// TIA Portal V17 export
// export: Created 2025-03-07T09:16:40.4760323Z, ExportSetting WithDefaults, DisplayName Totally Integrated Automation Portal, DisplayVersion V17 Update 8, DisplayName TIA Portal Openness, DisplayVersion V17 Update 8, DisplayName TIA Portal Version Control Interface, DisplayVersion V17, DisplayName SINAMICS Startdrive Advanced, DisplayVersion V17 SP2, DisplayName SINAMICS Startdrive G110M, G120, G120C, G120D, G120P, G115D, DisplayVersion V17 SP2, DisplayName SINAMICS Startdrive G130, G150, S120, S150, SINAMICS MV, S210, DisplayVersion V17 SP2, DisplayName STEP 7 Professional, DisplayVersion V17 Update 8, DisplayName SINUMERIK ONE STEP 7 Toolbox, DisplayVersion V17 Update 12, DisplayName SINUMERIK 840D sl STEP 7 Toolbox, DisplayVersion V17 Update 12, DisplayName STEP 7 Safety, DisplayVersion V17 Update 6, DisplayName WinCC Advanced, DisplayVersion V17 Update 8
FUNCTION "FC2431_FULL_DEPTHS_UNIT_02" : Void   // FC2431, LAD
{ S7_Optimized_Access := 'FALSE' }
AUTHOR : ETXETAR
VERSION : 1.0
// Fixture 1 and Fixture 3 will do Face A
// Fixture 2 and Fixture 4 will do Face B
// stored: AutoNumber false, IsIECCheckEnabled false, SetENOAutomatically false, UDAEnableTagReadback false
   VAR_TEMP   // added for the SCL form of the ladder/FBD networks
      _w1 : Bool;
   END_VAR
BEGIN

REGION Network 1: <<<<<<<<<<<<<<<<<<<<< UNIT 02 >>>>>>>>>>>>>>>>>>>>>
END_REGION

REGION Network 2: <<<<<<<<<<<<<<<<<<<< FIXTURE 1 >>>>>>>>>>>>>>>>>>>>
END_REGION

REGION Network 3: UNIT 02 FIXTURE 1 STATION 1 FULL DEPTH / FULL DEPTH 1 PULSE
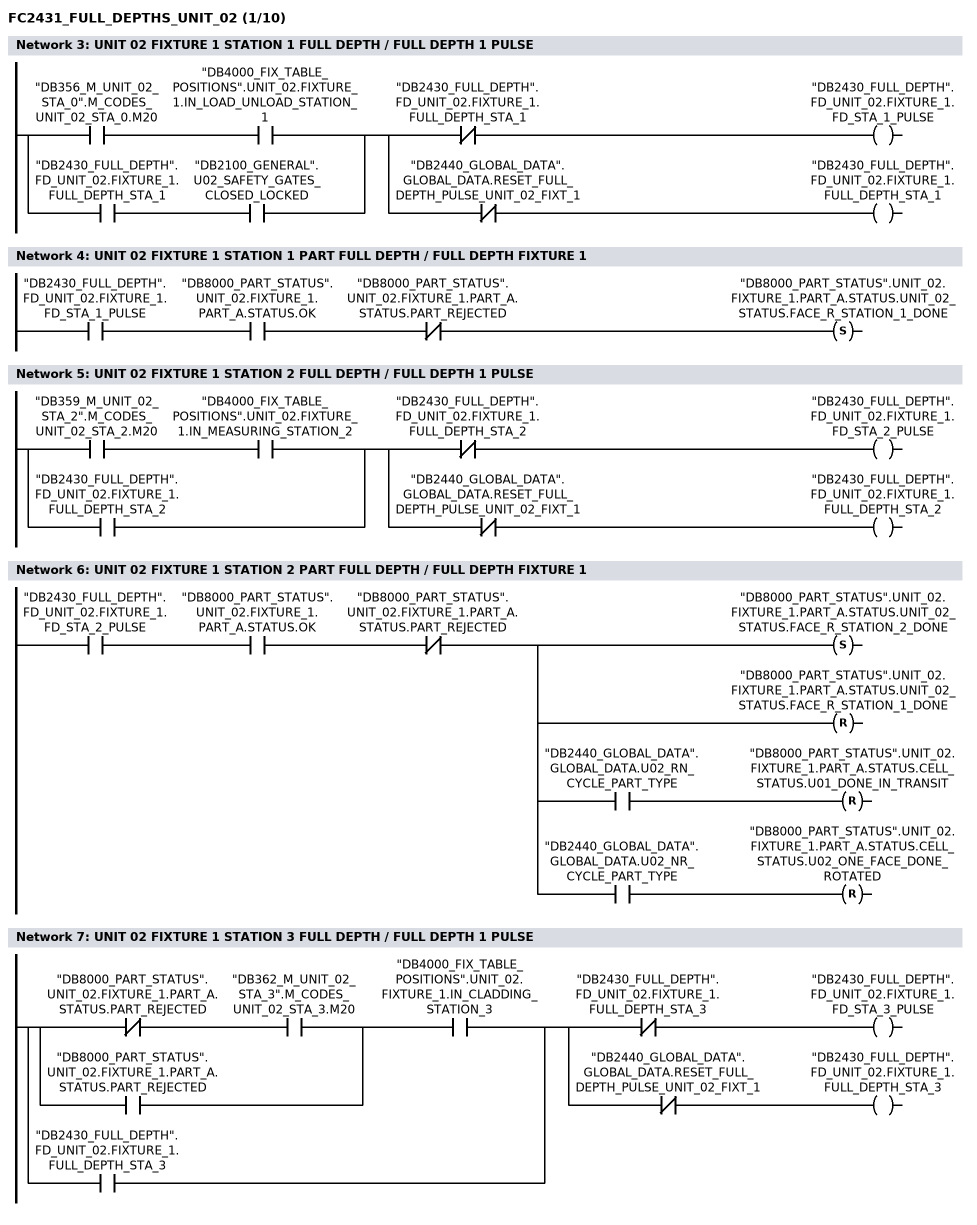
   RUNG wire#powerrail
      Contact( "DB356_M_UNIT_02_STA_0".M_CODES_UNIT_02_STA_0.M20 )
      Contact( "DB4000_FIX_TABLE_POSITIONS".UNIT_02.FIXTURE_1.IN_LOAD_UNLOAD_STATION_1 )
      wire#w1
      I_Contact( "DB2430_FULL_DEPTH".FD_UNIT_02.FIXTURE_1.FULL_DEPTH_STA_1 )
      Coil( "DB2430_FULL_DEPTH".FD_UNIT_02.FIXTURE_1.FD_STA_1_PULSE )
   END_RUNG
   RUNG wire#powerrail
      Contact( "DB2430_FULL_DEPTH".FD_UNIT_02.FIXTURE_1.FULL_DEPTH_STA_1 )
      Contact( "DB2100_GENERAL".U02_SAFETY_GATES_CLOSED_LOCKED )
   END_RUNG wire#w1
   RUNG wire#w1
      I_Contact( "DB2440_GLOBAL_DATA".GLOBAL_DATA.RESET_FULL_DEPTH_PULSE_UNIT_02_FIXT_1 )
      Coil( "DB2430_FULL_DEPTH".FD_UNIT_02.FIXTURE_1.FULL_DEPTH_STA_1 )
   END_RUNG
   // the same network as SCL:
   #_w1 := ("DB356_M_UNIT_02_STA_0".M_CODES_UNIT_02_STA_0.M20 AND "DB4000_FIX_TABLE_POSITIONS".UNIT_02.FIXTURE_1.IN_LOAD_UNLOAD_STATION_1) OR ("DB2430_FULL_DEPTH".FD_UNIT_02.FIXTURE_1.FULL_DEPTH_STA_1 AND "DB2100_GENERAL".U02_SAFETY_GATES_CLOSED_LOCKED);
   "DB2430_FULL_DEPTH".FD_UNIT_02.FIXTURE_1.FD_STA_1_PULSE := #_w1 AND NOT "DB2430_FULL_DEPTH".FD_UNIT_02.FIXTURE_1.FULL_DEPTH_STA_1;
   "DB2430_FULL_DEPTH".FD_UNIT_02.FIXTURE_1.FULL_DEPTH_STA_1 := #_w1 AND NOT "DB2440_GLOBAL_DATA".GLOBAL_DATA.RESET_FULL_DEPTH_PULSE_UNIT_02_FIXT_1;
END_REGION

REGION Network 4: UNIT 02 FIXTURE 1 STATION 1 PART FULL DEPTH / FULL DEPTH FIXTURE 1
   RUNG wire#powerrail
      Contact( "DB2430_FULL_DEPTH".FD_UNIT_02.FIXTURE_1.FD_STA_1_PULSE )
      Contact( "DB8000_PART_STATUS".UNIT_02.FIXTURE_1.PART_A.STATUS.OK )
      I_Contact( "DB8000_PART_STATUS".UNIT_02.FIXTURE_1.PART_A.STATUS.PART_REJECTED )
      S_Coil( "DB8000_PART_STATUS".UNIT_02.FIXTURE_1.PART_A.STATUS.UNIT_02_STATUS.FACE_R_STATION_1_DONE )
   END_RUNG
   // the same network as SCL:
   IF "DB2430_FULL_DEPTH".FD_UNIT_02.FIXTURE_1.FD_STA_1_PULSE AND "DB8000_PART_STATUS".UNIT_02.FIXTURE_1.PART_A.STATUS.OK AND NOT "DB8000_PART_STATUS".UNIT_02.FIXTURE_1.PART_A.STATUS.PART_REJECTED THEN
       "DB8000_PART_STATUS".UNIT_02.FIXTURE_1.PART_A.STATUS.UNIT_02_STATUS.FACE_R_STATION_1_DONE := TRUE;
   END_IF;
END_REGION

REGION Network 5: UNIT 02 FIXTURE 1 STATION 2 FULL DEPTH / FULL DEPTH 1 PULSE
   RUNG wire#powerrail
      Contact( "DB359_M_UNIT_02_STA_2".M_CODES_UNIT_02_STA_2.M20 )
      Contact( "DB4000_FIX_TABLE_POSITIONS".UNIT_02.FIXTURE_1.IN_MEASURING_STATION_2 )
      wire#w1
      I_Contact( "DB2430_FULL_DEPTH".FD_UNIT_02.FIXTURE_1.FULL_DEPTH_STA_2 )
      Coil( "DB2430_FULL_DEPTH".FD_UNIT_02.FIXTURE_1.FD_STA_2_PULSE )
   END_RUNG
   RUNG wire#powerrail
      Contact( "DB2430_FULL_DEPTH".FD_UNIT_02.FIXTURE_1.FULL_DEPTH_STA_2 )
   END_RUNG wire#w1
   RUNG wire#w1
      I_Contact( "DB2440_GLOBAL_DATA".GLOBAL_DATA.RESET_FULL_DEPTH_PULSE_UNIT_02_FIXT_1 )
      Coil( "DB2430_FULL_DEPTH".FD_UNIT_02.FIXTURE_1.FULL_DEPTH_STA_2 )
   END_RUNG
   // the same network as SCL:
   #_w1 := ("DB359_M_UNIT_02_STA_2".M_CODES_UNIT_02_STA_2.M20 AND "DB4000_FIX_TABLE_POSITIONS".UNIT_02.FIXTURE_1.IN_MEASURING_STATION_2) OR "DB2430_FULL_DEPTH".FD_UNIT_02.FIXTURE_1.FULL_DEPTH_STA_2;
   "DB2430_FULL_DEPTH".FD_UNIT_02.FIXTURE_1.FD_STA_2_PULSE := #_w1 AND NOT "DB2430_FULL_DEPTH".FD_UNIT_02.FIXTURE_1.FULL_DEPTH_STA_2;
   "DB2430_FULL_DEPTH".FD_UNIT_02.FIXTURE_1.FULL_DEPTH_STA_2 := #_w1 AND NOT "DB2440_GLOBAL_DATA".GLOBAL_DATA.RESET_FULL_DEPTH_PULSE_UNIT_02_FIXT_1;
END_REGION

REGION Network 6: UNIT 02 FIXTURE 1 STATION 2 PART FULL DEPTH / FULL DEPTH FIXTURE 1
   RUNG wire#powerrail
      Contact( "DB2430_FULL_DEPTH".FD_UNIT_02.FIXTURE_1.FD_STA_2_PULSE )
      Contact( "DB8000_PART_STATUS".UNIT_02.FIXTURE_1.PART_A.STATUS.OK )
      I_Contact( "DB8000_PART_STATUS".UNIT_02.FIXTURE_1.PART_A.STATUS.PART_REJECTED )
      wire#w1
      S_Coil( "DB8000_PART_STATUS".UNIT_02.FIXTURE_1.PART_A.STATUS.UNIT_02_STATUS.FACE_R_STATION_2_DONE )
   END_RUNG
   RUNG wire#w1
      R_Coil( "DB8000_PART_STATUS".UNIT_02.FIXTURE_1.PART_A.STATUS.UNIT_02_STATUS.FACE_R_STATION_1_DONE )
   END_RUNG
   RUNG wire#w1
      Contact( "DB2440_GLOBAL_DATA".GLOBAL_DATA.U02_RN_CYCLE_PART_TYPE )
      R_Coil( "DB8000_PART_STATUS".UNIT_02.FIXTURE_1.PART_A.STATUS.CELL_STATUS.U01_DONE_IN_TRANSIT )
   END_RUNG
   RUNG wire#w1
      Contact( "DB2440_GLOBAL_DATA".GLOBAL_DATA.U02_NR_CYCLE_PART_TYPE )
      R_Coil( "DB8000_PART_STATUS".UNIT_02.FIXTURE_1.PART_A.STATUS.CELL_STATUS.U02_ONE_FACE_DONE_ROTATED )
   END_RUNG
   // the same network as SCL:
   #_w1 := "DB2430_FULL_DEPTH".FD_UNIT_02.FIXTURE_1.FD_STA_2_PULSE AND "DB8000_PART_STATUS".UNIT_02.FIXTURE_1.PART_A.STATUS.OK AND NOT "DB8000_PART_STATUS".UNIT_02.FIXTURE_1.PART_A.STATUS.PART_REJECTED;
   IF #_w1 THEN
       "DB8000_PART_STATUS".UNIT_02.FIXTURE_1.PART_A.STATUS.UNIT_02_STATUS.FACE_R_STATION_2_DONE := TRUE;
       "DB8000_PART_STATUS".UNIT_02.FIXTURE_1.PART_A.STATUS.UNIT_02_STATUS.FACE_R_STATION_1_DONE := FALSE;
   END_IF;
   IF #_w1 AND "DB2440_GLOBAL_DATA".GLOBAL_DATA.U02_RN_CYCLE_PART_TYPE THEN
       "DB8000_PART_STATUS".UNIT_02.FIXTURE_1.PART_A.STATUS.CELL_STATUS.U01_DONE_IN_TRANSIT := FALSE;
   END_IF;
   IF #_w1 AND "DB2440_GLOBAL_DATA".GLOBAL_DATA.U02_NR_CYCLE_PART_TYPE THEN
       "DB8000_PART_STATUS".UNIT_02.FIXTURE_1.PART_A.STATUS.CELL_STATUS.U02_ONE_FACE_DONE_ROTATED := FALSE;
   END_IF;
END_REGION

REGION Network 7: UNIT 02 FIXTURE 1 STATION 3 FULL DEPTH / FULL DEPTH 1 PULSE
   RUNG wire#powerrail
      I_Contact( "DB8000_PART_STATUS".UNIT_02.FIXTURE_1.PART_A.STATUS.PART_REJECTED )
      Contact( "DB362_M_UNIT_02_STA_3".M_CODES_UNIT_02_STA_3.M20 )
      wire#w1
      Contact( "DB4000_FIX_TABLE_POSITIONS".UNIT_02.FIXTURE_1.IN_CLADDING_STATION_3 )
      wire#w2
      I_Contact( "DB2430_FULL_DEPTH".FD_UNIT_02.FIXTURE_1.FULL_DEPTH_STA_3 )
      Coil( "DB2430_FULL_DEPTH".FD_UNIT_02.FIXTURE_1.FD_STA_3_PULSE )
   END_RUNG
   RUNG wire#powerrail
      Contact( "DB8000_PART_STATUS".UNIT_02.FIXTURE_1.PART_A.STATUS.PART_REJECTED )
   END_RUNG wire#w1
   RUNG wire#powerrail
      Contact( "DB2430_FULL_DEPTH".FD_UNIT_02.FIXTURE_1.FULL_DEPTH_STA_3 )
   END_RUNG wire#w2
   RUNG wire#w2
      I_Contact( "DB2440_GLOBAL_DATA".GLOBAL_DATA.RESET_FULL_DEPTH_PULSE_UNIT_02_FIXT_1 )
      Coil( "DB2430_FULL_DEPTH".FD_UNIT_02.FIXTURE_1.FULL_DEPTH_STA_3 )
   END_RUNG
   // the same network as SCL:
   #_w1 := (((NOT "DB8000_PART_STATUS".UNIT_02.FIXTURE_1.PART_A.STATUS.PART_REJECTED AND "DB362_M_UNIT_02_STA_3".M_CODES_UNIT_02_STA_3.M20) OR "DB8000_PART_STATUS".UNIT_02.FIXTURE_1.PART_A.STATUS.PART_REJECTED) AND "DB4000_FIX_TABLE_POSITIONS".UNIT_02.FIXTURE_1.IN_CLADDING_STATION_3) OR "DB2430_FULL_DEPTH".FD_UNIT_02.FIXTURE_1.FULL_DEPTH_STA_3;
   "DB2430_FULL_DEPTH".FD_UNIT_02.FIXTURE_1.FD_STA_3_PULSE := #_w1 AND NOT "DB2430_FULL_DEPTH".FD_UNIT_02.FIXTURE_1.FULL_DEPTH_STA_3;
   "DB2430_FULL_DEPTH".FD_UNIT_02.FIXTURE_1.FULL_DEPTH_STA_3 := #_w1 AND NOT "DB2440_GLOBAL_DATA".GLOBAL_DATA.RESET_FULL_DEPTH_PULSE_UNIT_02_FIXT_1;
END_REGION

REGION Network 8: UNIT 02 FIXTURE 1 STATION 3 PART FULL DEPTH / FULL DEPTH FIXTURE 1
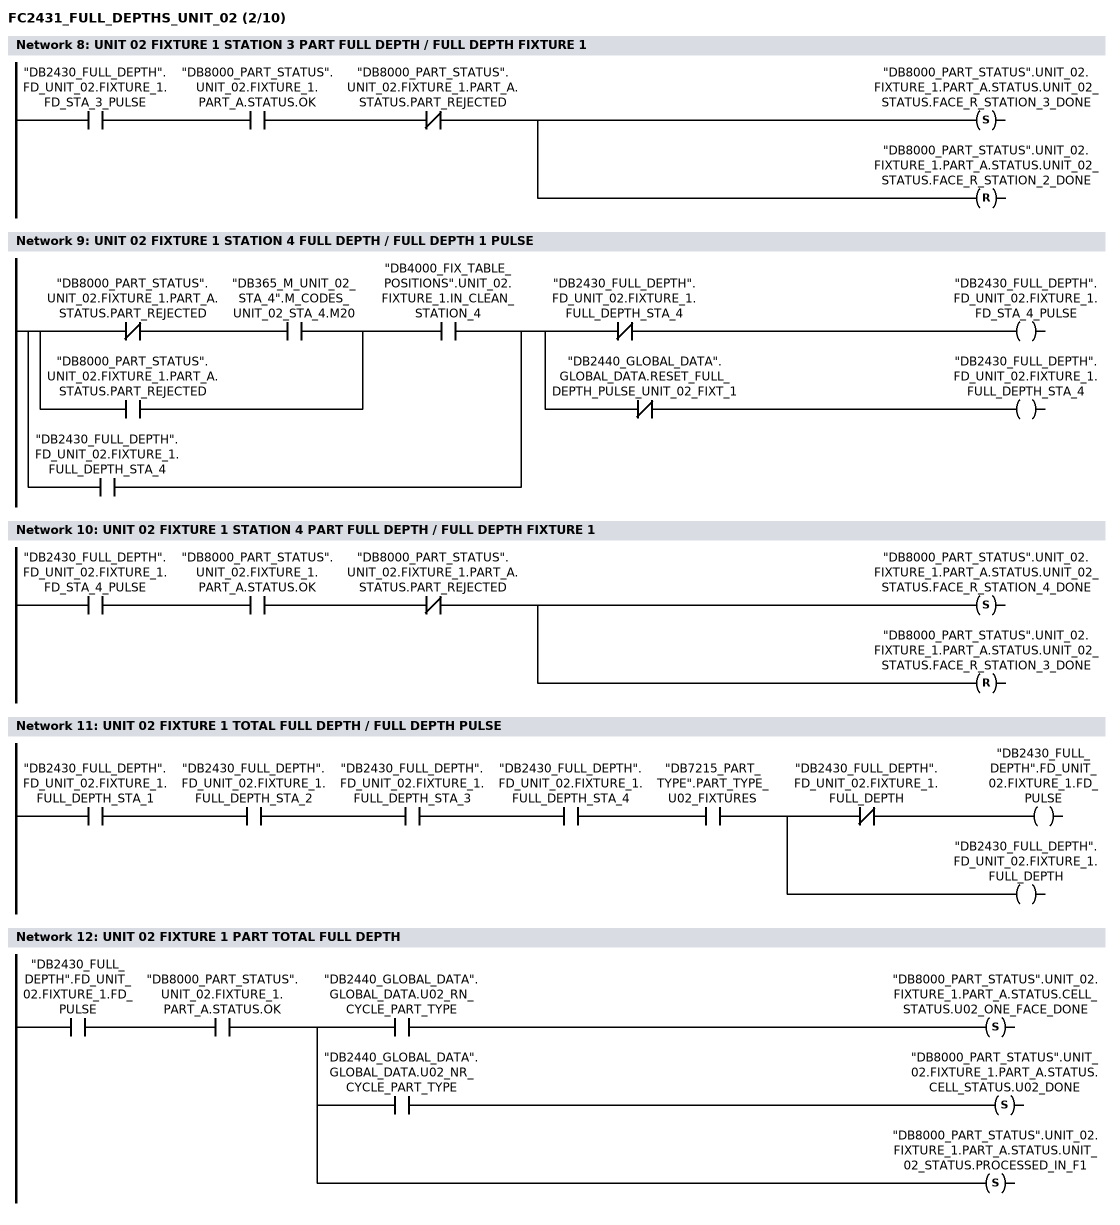
   RUNG wire#powerrail
      Contact( "DB2430_FULL_DEPTH".FD_UNIT_02.FIXTURE_1.FD_STA_3_PULSE )
      Contact( "DB8000_PART_STATUS".UNIT_02.FIXTURE_1.PART_A.STATUS.OK )
      I_Contact( "DB8000_PART_STATUS".UNIT_02.FIXTURE_1.PART_A.STATUS.PART_REJECTED )
      wire#w1
      S_Coil( "DB8000_PART_STATUS".UNIT_02.FIXTURE_1.PART_A.STATUS.UNIT_02_STATUS.FACE_R_STATION_3_DONE )
   END_RUNG
   RUNG wire#w1
      R_Coil( "DB8000_PART_STATUS".UNIT_02.FIXTURE_1.PART_A.STATUS.UNIT_02_STATUS.FACE_R_STATION_2_DONE )
   END_RUNG
   // the same network as SCL:
   IF "DB2430_FULL_DEPTH".FD_UNIT_02.FIXTURE_1.FD_STA_3_PULSE AND "DB8000_PART_STATUS".UNIT_02.FIXTURE_1.PART_A.STATUS.OK AND NOT "DB8000_PART_STATUS".UNIT_02.FIXTURE_1.PART_A.STATUS.PART_REJECTED THEN
       "DB8000_PART_STATUS".UNIT_02.FIXTURE_1.PART_A.STATUS.UNIT_02_STATUS.FACE_R_STATION_3_DONE := TRUE;
       "DB8000_PART_STATUS".UNIT_02.FIXTURE_1.PART_A.STATUS.UNIT_02_STATUS.FACE_R_STATION_2_DONE := FALSE;
   END_IF;
END_REGION

REGION Network 9: UNIT 02 FIXTURE 1 STATION 4 FULL DEPTH / FULL DEPTH 1 PULSE
   RUNG wire#powerrail
      I_Contact( "DB8000_PART_STATUS".UNIT_02.FIXTURE_1.PART_A.STATUS.PART_REJECTED )
      Contact( "DB365_M_UNIT_02_STA_4".M_CODES_UNIT_02_STA_4.M20 )
      wire#w1
      Contact( "DB4000_FIX_TABLE_POSITIONS".UNIT_02.FIXTURE_1.IN_CLEAN_STATION_4 )
      wire#w2
      I_Contact( "DB2430_FULL_DEPTH".FD_UNIT_02.FIXTURE_1.FULL_DEPTH_STA_4 )
      Coil( "DB2430_FULL_DEPTH".FD_UNIT_02.FIXTURE_1.FD_STA_4_PULSE )
   END_RUNG
   RUNG wire#powerrail
      Contact( "DB8000_PART_STATUS".UNIT_02.FIXTURE_1.PART_A.STATUS.PART_REJECTED )
   END_RUNG wire#w1
   RUNG wire#powerrail
      Contact( "DB2430_FULL_DEPTH".FD_UNIT_02.FIXTURE_1.FULL_DEPTH_STA_4 )
   END_RUNG wire#w2
   RUNG wire#w2
      I_Contact( "DB2440_GLOBAL_DATA".GLOBAL_DATA.RESET_FULL_DEPTH_PULSE_UNIT_02_FIXT_1 )
      Coil( "DB2430_FULL_DEPTH".FD_UNIT_02.FIXTURE_1.FULL_DEPTH_STA_4 )
   END_RUNG
   // the same network as SCL:
   #_w1 := (((NOT "DB8000_PART_STATUS".UNIT_02.FIXTURE_1.PART_A.STATUS.PART_REJECTED AND "DB365_M_UNIT_02_STA_4".M_CODES_UNIT_02_STA_4.M20) OR "DB8000_PART_STATUS".UNIT_02.FIXTURE_1.PART_A.STATUS.PART_REJECTED) AND "DB4000_FIX_TABLE_POSITIONS".UNIT_02.FIXTURE_1.IN_CLEAN_STATION_4) OR "DB2430_FULL_DEPTH".FD_UNIT_02.FIXTURE_1.FULL_DEPTH_STA_4;
   "DB2430_FULL_DEPTH".FD_UNIT_02.FIXTURE_1.FD_STA_4_PULSE := #_w1 AND NOT "DB2430_FULL_DEPTH".FD_UNIT_02.FIXTURE_1.FULL_DEPTH_STA_4;
   "DB2430_FULL_DEPTH".FD_UNIT_02.FIXTURE_1.FULL_DEPTH_STA_4 := #_w1 AND NOT "DB2440_GLOBAL_DATA".GLOBAL_DATA.RESET_FULL_DEPTH_PULSE_UNIT_02_FIXT_1;
END_REGION

REGION Network 10: UNIT 02 FIXTURE 1 STATION 4 PART FULL DEPTH / FULL DEPTH FIXTURE 1
   RUNG wire#powerrail
      Contact( "DB2430_FULL_DEPTH".FD_UNIT_02.FIXTURE_1.FD_STA_4_PULSE )
      Contact( "DB8000_PART_STATUS".UNIT_02.FIXTURE_1.PART_A.STATUS.OK )
      I_Contact( "DB8000_PART_STATUS".UNIT_02.FIXTURE_1.PART_A.STATUS.PART_REJECTED )
      wire#w1
      S_Coil( "DB8000_PART_STATUS".UNIT_02.FIXTURE_1.PART_A.STATUS.UNIT_02_STATUS.FACE_R_STATION_4_DONE )
   END_RUNG
   RUNG wire#w1
      R_Coil( "DB8000_PART_STATUS".UNIT_02.FIXTURE_1.PART_A.STATUS.UNIT_02_STATUS.FACE_R_STATION_3_DONE )
   END_RUNG
   // the same network as SCL:
   IF "DB2430_FULL_DEPTH".FD_UNIT_02.FIXTURE_1.FD_STA_4_PULSE AND "DB8000_PART_STATUS".UNIT_02.FIXTURE_1.PART_A.STATUS.OK AND NOT "DB8000_PART_STATUS".UNIT_02.FIXTURE_1.PART_A.STATUS.PART_REJECTED THEN
       "DB8000_PART_STATUS".UNIT_02.FIXTURE_1.PART_A.STATUS.UNIT_02_STATUS.FACE_R_STATION_4_DONE := TRUE;
       "DB8000_PART_STATUS".UNIT_02.FIXTURE_1.PART_A.STATUS.UNIT_02_STATUS.FACE_R_STATION_3_DONE := FALSE;
   END_IF;
END_REGION

REGION Network 11: UNIT 02 FIXTURE 1 TOTAL FULL DEPTH / FULL DEPTH PULSE
   RUNG wire#powerrail
      Contact( "DB2430_FULL_DEPTH".FD_UNIT_02.FIXTURE_1.FULL_DEPTH_STA_1 )
      Contact( "DB2430_FULL_DEPTH".FD_UNIT_02.FIXTURE_1.FULL_DEPTH_STA_2 )
      Contact( "DB2430_FULL_DEPTH".FD_UNIT_02.FIXTURE_1.FULL_DEPTH_STA_3 )
      Contact( "DB2430_FULL_DEPTH".FD_UNIT_02.FIXTURE_1.FULL_DEPTH_STA_4 )
      Contact( "DB7215_PART_TYPE".PART_TYPE_U02_FIXTURES )
      wire#w1
      I_Contact( "DB2430_FULL_DEPTH".FD_UNIT_02.FIXTURE_1.FULL_DEPTH )
      Coil( "DB2430_FULL_DEPTH".FD_UNIT_02.FIXTURE_1.FD_PULSE )
   END_RUNG
   RUNG wire#w1
      Coil( "DB2430_FULL_DEPTH".FD_UNIT_02.FIXTURE_1.FULL_DEPTH )
   END_RUNG
   // the same network as SCL:
   #_w1 := "DB2430_FULL_DEPTH".FD_UNIT_02.FIXTURE_1.FULL_DEPTH_STA_1 AND "DB2430_FULL_DEPTH".FD_UNIT_02.FIXTURE_1.FULL_DEPTH_STA_2 AND "DB2430_FULL_DEPTH".FD_UNIT_02.FIXTURE_1.FULL_DEPTH_STA_3 AND "DB2430_FULL_DEPTH".FD_UNIT_02.FIXTURE_1.FULL_DEPTH_STA_4 AND "DB7215_PART_TYPE".PART_TYPE_U02_FIXTURES;
   "DB2430_FULL_DEPTH".FD_UNIT_02.FIXTURE_1.FD_PULSE := #_w1 AND NOT "DB2430_FULL_DEPTH".FD_UNIT_02.FIXTURE_1.FULL_DEPTH;
   "DB2430_FULL_DEPTH".FD_UNIT_02.FIXTURE_1.FULL_DEPTH := #_w1;
END_REGION

REGION Network 12: UNIT 02 FIXTURE 1 PART TOTAL FULL DEPTH
   RUNG wire#powerrail
      Contact( "DB2430_FULL_DEPTH".FD_UNIT_02.FIXTURE_1.FD_PULSE )
      Contact( "DB8000_PART_STATUS".UNIT_02.FIXTURE_1.PART_A.STATUS.OK )
      wire#w1
      Contact( "DB2440_GLOBAL_DATA".GLOBAL_DATA.U02_RN_CYCLE_PART_TYPE )
      S_Coil( "DB8000_PART_STATUS".UNIT_02.FIXTURE_1.PART_A.STATUS.CELL_STATUS.U02_ONE_FACE_DONE )
   END_RUNG
   RUNG wire#w1
      Contact( "DB2440_GLOBAL_DATA".GLOBAL_DATA.U02_NR_CYCLE_PART_TYPE )
      S_Coil( "DB8000_PART_STATUS".UNIT_02.FIXTURE_1.PART_A.STATUS.CELL_STATUS.U02_DONE )
   END_RUNG
   RUNG wire#w1
      S_Coil( "DB8000_PART_STATUS".UNIT_02.FIXTURE_1.PART_A.STATUS.UNIT_02_STATUS.PROCESSED_IN_F1 )
   END_RUNG
   // the same network as SCL:
   #_w1 := "DB2430_FULL_DEPTH".FD_UNIT_02.FIXTURE_1.FD_PULSE AND "DB8000_PART_STATUS".UNIT_02.FIXTURE_1.PART_A.STATUS.OK;
   IF #_w1 AND "DB2440_GLOBAL_DATA".GLOBAL_DATA.U02_RN_CYCLE_PART_TYPE THEN
       "DB8000_PART_STATUS".UNIT_02.FIXTURE_1.PART_A.STATUS.CELL_STATUS.U02_ONE_FACE_DONE := TRUE;
   END_IF;
   IF #_w1 AND "DB2440_GLOBAL_DATA".GLOBAL_DATA.U02_NR_CYCLE_PART_TYPE THEN
       "DB8000_PART_STATUS".UNIT_02.FIXTURE_1.PART_A.STATUS.CELL_STATUS.U02_DONE := TRUE;
   END_IF;
   IF #_w1 THEN
       "DB8000_PART_STATUS".UNIT_02.FIXTURE_1.PART_A.STATUS.UNIT_02_STATUS.PROCESSED_IN_F1 := TRUE;
   END_IF;
END_REGION

REGION Network 13: UNIT 02 FIXTURE 1 PART REJECTED / PART HAS BEEN REJECTED
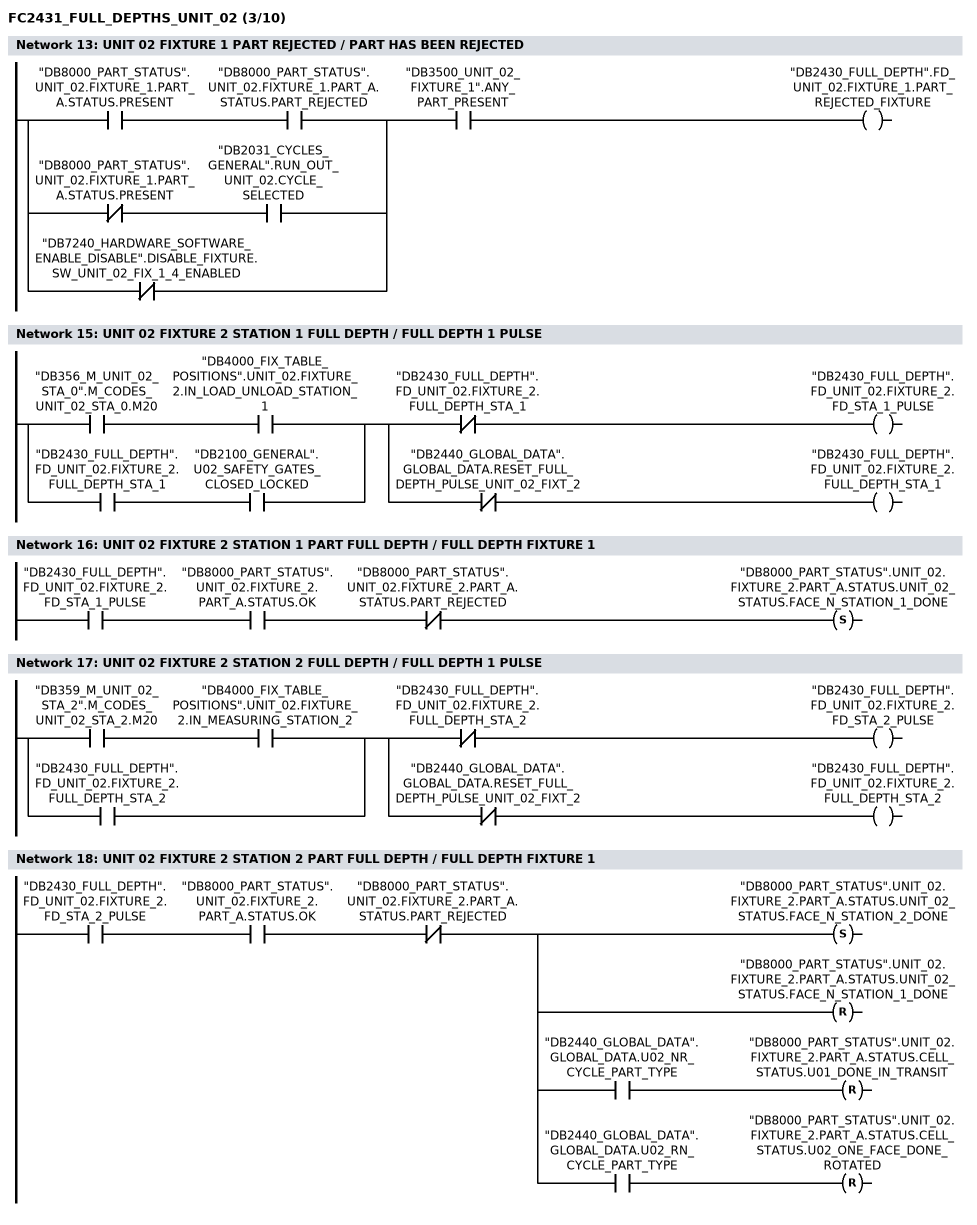
   RUNG wire#powerrail
      Contact( "DB8000_PART_STATUS".UNIT_02.FIXTURE_1.PART_A.STATUS.PRESENT )
      Contact( "DB8000_PART_STATUS".UNIT_02.FIXTURE_1.PART_A.STATUS.PART_REJECTED )
      wire#w1
      Contact( "DB3500_UNIT_02_FIXTURE_1".ANY_PART_PRESENT )
      Coil( "DB2430_FULL_DEPTH".FD_UNIT_02.FIXTURE_1.PART_REJECTED_FIXTURE )
   END_RUNG
   RUNG wire#powerrail
      I_Contact( "DB8000_PART_STATUS".UNIT_02.FIXTURE_1.PART_A.STATUS.PRESENT )
      Contact( "DB2031_CYCLES_GENERAL".RUN_OUT_UNIT_02.CYCLE_SELECTED )
   END_RUNG wire#w1
   RUNG wire#powerrail
      I_Contact( "DB7240_HARDWARE_SOFTWARE_ENABLE_DISABLE".DISABLE_FIXTURE.SW_UNIT_02_FIX_1_4_ENABLED )
   END_RUNG wire#w1
   // the same network as SCL:
   "DB2430_FULL_DEPTH".FD_UNIT_02.FIXTURE_1.PART_REJECTED_FIXTURE := (("DB8000_PART_STATUS".UNIT_02.FIXTURE_1.PART_A.STATUS.PRESENT AND "DB8000_PART_STATUS".UNIT_02.FIXTURE_1.PART_A.STATUS.PART_REJECTED) OR (NOT "DB8000_PART_STATUS".UNIT_02.FIXTURE_1.PART_A.STATUS.PRESENT AND "DB2031_CYCLES_GENERAL".RUN_OUT_UNIT_02.CYCLE_SELECTED) OR NOT "DB7240_HARDWARE_SOFTWARE_ENABLE_DISABLE".DISABLE_FIXTURE.SW_UNIT_02_FIX_1_4_ENABLED) AND "DB3500_UNIT_02_FIXTURE_1".ANY_PART_PRESENT;
END_REGION

REGION Network 14: <<<<<<<<<<<<<<<<<<<< FIXTURE 2 >>>>>>>>>>>>>>>>>>>>
END_REGION

REGION Network 15: UNIT 02 FIXTURE 2 STATION 1 FULL DEPTH / FULL DEPTH 1 PULSE
   RUNG wire#powerrail
      Contact( "DB356_M_UNIT_02_STA_0".M_CODES_UNIT_02_STA_0.M20 )
      Contact( "DB4000_FIX_TABLE_POSITIONS".UNIT_02.FIXTURE_2.IN_LOAD_UNLOAD_STATION_1 )
      wire#w1
      I_Contact( "DB2430_FULL_DEPTH".FD_UNIT_02.FIXTURE_2.FULL_DEPTH_STA_1 )
      Coil( "DB2430_FULL_DEPTH".FD_UNIT_02.FIXTURE_2.FD_STA_1_PULSE )
   END_RUNG
   RUNG wire#powerrail
      Contact( "DB2430_FULL_DEPTH".FD_UNIT_02.FIXTURE_2.FULL_DEPTH_STA_1 )
      Contact( "DB2100_GENERAL".U02_SAFETY_GATES_CLOSED_LOCKED )
   END_RUNG wire#w1
   RUNG wire#w1
      I_Contact( "DB2440_GLOBAL_DATA".GLOBAL_DATA.RESET_FULL_DEPTH_PULSE_UNIT_02_FIXT_2 )
      Coil( "DB2430_FULL_DEPTH".FD_UNIT_02.FIXTURE_2.FULL_DEPTH_STA_1 )
   END_RUNG
   // the same network as SCL:
   #_w1 := ("DB356_M_UNIT_02_STA_0".M_CODES_UNIT_02_STA_0.M20 AND "DB4000_FIX_TABLE_POSITIONS".UNIT_02.FIXTURE_2.IN_LOAD_UNLOAD_STATION_1) OR ("DB2430_FULL_DEPTH".FD_UNIT_02.FIXTURE_2.FULL_DEPTH_STA_1 AND "DB2100_GENERAL".U02_SAFETY_GATES_CLOSED_LOCKED);
   "DB2430_FULL_DEPTH".FD_UNIT_02.FIXTURE_2.FD_STA_1_PULSE := #_w1 AND NOT "DB2430_FULL_DEPTH".FD_UNIT_02.FIXTURE_2.FULL_DEPTH_STA_1;
   "DB2430_FULL_DEPTH".FD_UNIT_02.FIXTURE_2.FULL_DEPTH_STA_1 := #_w1 AND NOT "DB2440_GLOBAL_DATA".GLOBAL_DATA.RESET_FULL_DEPTH_PULSE_UNIT_02_FIXT_2;
END_REGION

REGION Network 16: UNIT 02 FIXTURE 2 STATION 1 PART FULL DEPTH / FULL DEPTH FIXTURE 1
   RUNG wire#powerrail
      Contact( "DB2430_FULL_DEPTH".FD_UNIT_02.FIXTURE_2.FD_STA_1_PULSE )
      Contact( "DB8000_PART_STATUS".UNIT_02.FIXTURE_2.PART_A.STATUS.OK )
      I_Contact( "DB8000_PART_STATUS".UNIT_02.FIXTURE_2.PART_A.STATUS.PART_REJECTED )
      S_Coil( "DB8000_PART_STATUS".UNIT_02.FIXTURE_2.PART_A.STATUS.UNIT_02_STATUS.FACE_N_STATION_1_DONE )
   END_RUNG
   // the same network as SCL:
   IF "DB2430_FULL_DEPTH".FD_UNIT_02.FIXTURE_2.FD_STA_1_PULSE AND "DB8000_PART_STATUS".UNIT_02.FIXTURE_2.PART_A.STATUS.OK AND NOT "DB8000_PART_STATUS".UNIT_02.FIXTURE_2.PART_A.STATUS.PART_REJECTED THEN
       "DB8000_PART_STATUS".UNIT_02.FIXTURE_2.PART_A.STATUS.UNIT_02_STATUS.FACE_N_STATION_1_DONE := TRUE;
   END_IF;
END_REGION

REGION Network 17: UNIT 02 FIXTURE 2 STATION 2 FULL DEPTH / FULL DEPTH 1 PULSE
   RUNG wire#powerrail
      Contact( "DB359_M_UNIT_02_STA_2".M_CODES_UNIT_02_STA_2.M20 )
      Contact( "DB4000_FIX_TABLE_POSITIONS".UNIT_02.FIXTURE_2.IN_MEASURING_STATION_2 )
      wire#w1
      I_Contact( "DB2430_FULL_DEPTH".FD_UNIT_02.FIXTURE_2.FULL_DEPTH_STA_2 )
      Coil( "DB2430_FULL_DEPTH".FD_UNIT_02.FIXTURE_2.FD_STA_2_PULSE )
   END_RUNG
   RUNG wire#powerrail
      Contact( "DB2430_FULL_DEPTH".FD_UNIT_02.FIXTURE_2.FULL_DEPTH_STA_2 )
   END_RUNG wire#w1
   RUNG wire#w1
      I_Contact( "DB2440_GLOBAL_DATA".GLOBAL_DATA.RESET_FULL_DEPTH_PULSE_UNIT_02_FIXT_2 )
      Coil( "DB2430_FULL_DEPTH".FD_UNIT_02.FIXTURE_2.FULL_DEPTH_STA_2 )
   END_RUNG
   // the same network as SCL:
   #_w1 := ("DB359_M_UNIT_02_STA_2".M_CODES_UNIT_02_STA_2.M20 AND "DB4000_FIX_TABLE_POSITIONS".UNIT_02.FIXTURE_2.IN_MEASURING_STATION_2) OR "DB2430_FULL_DEPTH".FD_UNIT_02.FIXTURE_2.FULL_DEPTH_STA_2;
   "DB2430_FULL_DEPTH".FD_UNIT_02.FIXTURE_2.FD_STA_2_PULSE := #_w1 AND NOT "DB2430_FULL_DEPTH".FD_UNIT_02.FIXTURE_2.FULL_DEPTH_STA_2;
   "DB2430_FULL_DEPTH".FD_UNIT_02.FIXTURE_2.FULL_DEPTH_STA_2 := #_w1 AND NOT "DB2440_GLOBAL_DATA".GLOBAL_DATA.RESET_FULL_DEPTH_PULSE_UNIT_02_FIXT_2;
END_REGION

REGION Network 18: UNIT 02 FIXTURE 2 STATION 2 PART FULL DEPTH / FULL DEPTH FIXTURE 1
   RUNG wire#powerrail
      Contact( "DB2430_FULL_DEPTH".FD_UNIT_02.FIXTURE_2.FD_STA_2_PULSE )
      Contact( "DB8000_PART_STATUS".UNIT_02.FIXTURE_2.PART_A.STATUS.OK )
      I_Contact( "DB8000_PART_STATUS".UNIT_02.FIXTURE_2.PART_A.STATUS.PART_REJECTED )
      wire#w1
      S_Coil( "DB8000_PART_STATUS".UNIT_02.FIXTURE_2.PART_A.STATUS.UNIT_02_STATUS.FACE_N_STATION_2_DONE )
   END_RUNG
   RUNG wire#w1
      R_Coil( "DB8000_PART_STATUS".UNIT_02.FIXTURE_2.PART_A.STATUS.UNIT_02_STATUS.FACE_N_STATION_1_DONE )
   END_RUNG
   RUNG wire#w1
      Contact( "DB2440_GLOBAL_DATA".GLOBAL_DATA.U02_NR_CYCLE_PART_TYPE )
      R_Coil( "DB8000_PART_STATUS".UNIT_02.FIXTURE_2.PART_A.STATUS.CELL_STATUS.U01_DONE_IN_TRANSIT )
   END_RUNG
   RUNG wire#w1
      Contact( "DB2440_GLOBAL_DATA".GLOBAL_DATA.U02_RN_CYCLE_PART_TYPE )
      R_Coil( "DB8000_PART_STATUS".UNIT_02.FIXTURE_2.PART_A.STATUS.CELL_STATUS.U02_ONE_FACE_DONE_ROTATED )
   END_RUNG
   // the same network as SCL:
   #_w1 := "DB2430_FULL_DEPTH".FD_UNIT_02.FIXTURE_2.FD_STA_2_PULSE AND "DB8000_PART_STATUS".UNIT_02.FIXTURE_2.PART_A.STATUS.OK AND NOT "DB8000_PART_STATUS".UNIT_02.FIXTURE_2.PART_A.STATUS.PART_REJECTED;
   IF #_w1 THEN
       "DB8000_PART_STATUS".UNIT_02.FIXTURE_2.PART_A.STATUS.UNIT_02_STATUS.FACE_N_STATION_2_DONE := TRUE;
       "DB8000_PART_STATUS".UNIT_02.FIXTURE_2.PART_A.STATUS.UNIT_02_STATUS.FACE_N_STATION_1_DONE := FALSE;
   END_IF;
   IF #_w1 AND "DB2440_GLOBAL_DATA".GLOBAL_DATA.U02_NR_CYCLE_PART_TYPE THEN
       "DB8000_PART_STATUS".UNIT_02.FIXTURE_2.PART_A.STATUS.CELL_STATUS.U01_DONE_IN_TRANSIT := FALSE;
   END_IF;
   IF #_w1 AND "DB2440_GLOBAL_DATA".GLOBAL_DATA.U02_RN_CYCLE_PART_TYPE THEN
       "DB8000_PART_STATUS".UNIT_02.FIXTURE_2.PART_A.STATUS.CELL_STATUS.U02_ONE_FACE_DONE_ROTATED := FALSE;
   END_IF;
END_REGION

REGION Network 19: UNIT 02 FIXTURE 2 STATION 3 FULL DEPTH / FULL DEPTH 1 PULSE
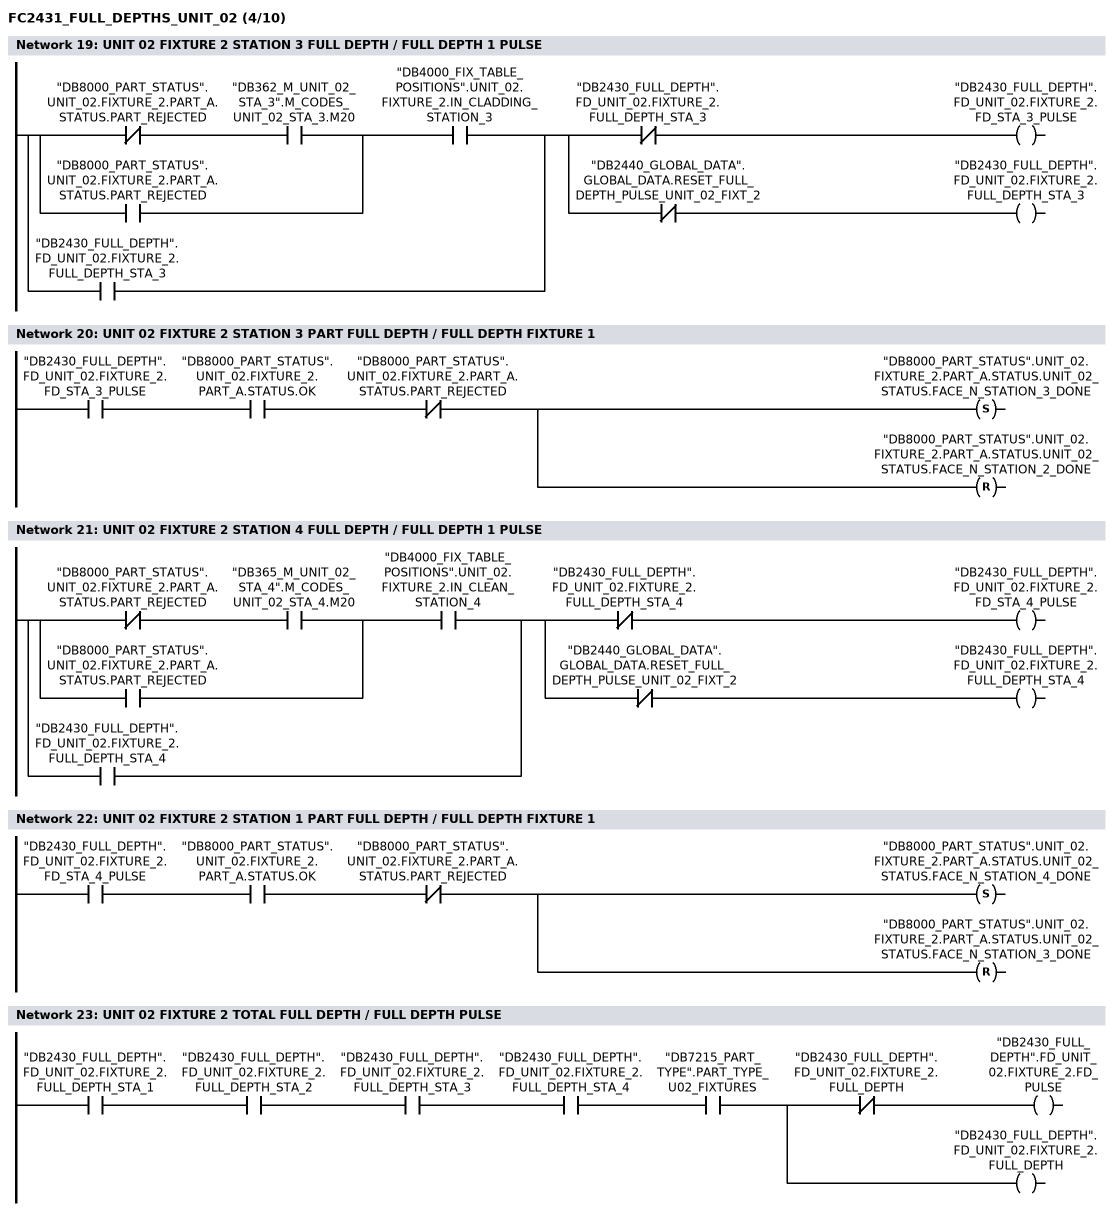
   RUNG wire#powerrail
      I_Contact( "DB8000_PART_STATUS".UNIT_02.FIXTURE_2.PART_A.STATUS.PART_REJECTED )
      Contact( "DB362_M_UNIT_02_STA_3".M_CODES_UNIT_02_STA_3.M20 )
      wire#w1
      Contact( "DB4000_FIX_TABLE_POSITIONS".UNIT_02.FIXTURE_2.IN_CLADDING_STATION_3 )
      wire#w2
      I_Contact( "DB2430_FULL_DEPTH".FD_UNIT_02.FIXTURE_2.FULL_DEPTH_STA_3 )
      Coil( "DB2430_FULL_DEPTH".FD_UNIT_02.FIXTURE_2.FD_STA_3_PULSE )
   END_RUNG
   RUNG wire#powerrail
      Contact( "DB8000_PART_STATUS".UNIT_02.FIXTURE_2.PART_A.STATUS.PART_REJECTED )
   END_RUNG wire#w1
   RUNG wire#powerrail
      Contact( "DB2430_FULL_DEPTH".FD_UNIT_02.FIXTURE_2.FULL_DEPTH_STA_3 )
   END_RUNG wire#w2
   RUNG wire#w2
      I_Contact( "DB2440_GLOBAL_DATA".GLOBAL_DATA.RESET_FULL_DEPTH_PULSE_UNIT_02_FIXT_2 )
      Coil( "DB2430_FULL_DEPTH".FD_UNIT_02.FIXTURE_2.FULL_DEPTH_STA_3 )
   END_RUNG
   // the same network as SCL:
   #_w1 := (((NOT "DB8000_PART_STATUS".UNIT_02.FIXTURE_2.PART_A.STATUS.PART_REJECTED AND "DB362_M_UNIT_02_STA_3".M_CODES_UNIT_02_STA_3.M20) OR "DB8000_PART_STATUS".UNIT_02.FIXTURE_2.PART_A.STATUS.PART_REJECTED) AND "DB4000_FIX_TABLE_POSITIONS".UNIT_02.FIXTURE_2.IN_CLADDING_STATION_3) OR "DB2430_FULL_DEPTH".FD_UNIT_02.FIXTURE_2.FULL_DEPTH_STA_3;
   "DB2430_FULL_DEPTH".FD_UNIT_02.FIXTURE_2.FD_STA_3_PULSE := #_w1 AND NOT "DB2430_FULL_DEPTH".FD_UNIT_02.FIXTURE_2.FULL_DEPTH_STA_3;
   "DB2430_FULL_DEPTH".FD_UNIT_02.FIXTURE_2.FULL_DEPTH_STA_3 := #_w1 AND NOT "DB2440_GLOBAL_DATA".GLOBAL_DATA.RESET_FULL_DEPTH_PULSE_UNIT_02_FIXT_2;
END_REGION

REGION Network 20: UNIT 02 FIXTURE 2 STATION 3 PART FULL DEPTH / FULL DEPTH FIXTURE 1
   RUNG wire#powerrail
      Contact( "DB2430_FULL_DEPTH".FD_UNIT_02.FIXTURE_2.FD_STA_3_PULSE )
      Contact( "DB8000_PART_STATUS".UNIT_02.FIXTURE_2.PART_A.STATUS.OK )
      I_Contact( "DB8000_PART_STATUS".UNIT_02.FIXTURE_2.PART_A.STATUS.PART_REJECTED )
      wire#w1
      S_Coil( "DB8000_PART_STATUS".UNIT_02.FIXTURE_2.PART_A.STATUS.UNIT_02_STATUS.FACE_N_STATION_3_DONE )
   END_RUNG
   RUNG wire#w1
      R_Coil( "DB8000_PART_STATUS".UNIT_02.FIXTURE_2.PART_A.STATUS.UNIT_02_STATUS.FACE_N_STATION_2_DONE )
   END_RUNG
   // the same network as SCL:
   IF "DB2430_FULL_DEPTH".FD_UNIT_02.FIXTURE_2.FD_STA_3_PULSE AND "DB8000_PART_STATUS".UNIT_02.FIXTURE_2.PART_A.STATUS.OK AND NOT "DB8000_PART_STATUS".UNIT_02.FIXTURE_2.PART_A.STATUS.PART_REJECTED THEN
       "DB8000_PART_STATUS".UNIT_02.FIXTURE_2.PART_A.STATUS.UNIT_02_STATUS.FACE_N_STATION_3_DONE := TRUE;
       "DB8000_PART_STATUS".UNIT_02.FIXTURE_2.PART_A.STATUS.UNIT_02_STATUS.FACE_N_STATION_2_DONE := FALSE;
   END_IF;
END_REGION

REGION Network 21: UNIT 02 FIXTURE 2 STATION 4 FULL DEPTH / FULL DEPTH 1 PULSE
   RUNG wire#powerrail
      I_Contact( "DB8000_PART_STATUS".UNIT_02.FIXTURE_2.PART_A.STATUS.PART_REJECTED )
      Contact( "DB365_M_UNIT_02_STA_4".M_CODES_UNIT_02_STA_4.M20 )
      wire#w1
      Contact( "DB4000_FIX_TABLE_POSITIONS".UNIT_02.FIXTURE_2.IN_CLEAN_STATION_4 )
      wire#w2
      I_Contact( "DB2430_FULL_DEPTH".FD_UNIT_02.FIXTURE_2.FULL_DEPTH_STA_4 )
      Coil( "DB2430_FULL_DEPTH".FD_UNIT_02.FIXTURE_2.FD_STA_4_PULSE )
   END_RUNG
   RUNG wire#powerrail
      Contact( "DB8000_PART_STATUS".UNIT_02.FIXTURE_2.PART_A.STATUS.PART_REJECTED )
   END_RUNG wire#w1
   RUNG wire#powerrail
      Contact( "DB2430_FULL_DEPTH".FD_UNIT_02.FIXTURE_2.FULL_DEPTH_STA_4 )
   END_RUNG wire#w2
   RUNG wire#w2
      I_Contact( "DB2440_GLOBAL_DATA".GLOBAL_DATA.RESET_FULL_DEPTH_PULSE_UNIT_02_FIXT_2 )
      Coil( "DB2430_FULL_DEPTH".FD_UNIT_02.FIXTURE_2.FULL_DEPTH_STA_4 )
   END_RUNG
   // the same network as SCL:
   #_w1 := (((NOT "DB8000_PART_STATUS".UNIT_02.FIXTURE_2.PART_A.STATUS.PART_REJECTED AND "DB365_M_UNIT_02_STA_4".M_CODES_UNIT_02_STA_4.M20) OR "DB8000_PART_STATUS".UNIT_02.FIXTURE_2.PART_A.STATUS.PART_REJECTED) AND "DB4000_FIX_TABLE_POSITIONS".UNIT_02.FIXTURE_2.IN_CLEAN_STATION_4) OR "DB2430_FULL_DEPTH".FD_UNIT_02.FIXTURE_2.FULL_DEPTH_STA_4;
   "DB2430_FULL_DEPTH".FD_UNIT_02.FIXTURE_2.FD_STA_4_PULSE := #_w1 AND NOT "DB2430_FULL_DEPTH".FD_UNIT_02.FIXTURE_2.FULL_DEPTH_STA_4;
   "DB2430_FULL_DEPTH".FD_UNIT_02.FIXTURE_2.FULL_DEPTH_STA_4 := #_w1 AND NOT "DB2440_GLOBAL_DATA".GLOBAL_DATA.RESET_FULL_DEPTH_PULSE_UNIT_02_FIXT_2;
END_REGION

REGION Network 22: UNIT 02 FIXTURE 2 STATION 1 PART FULL DEPTH / FULL DEPTH FIXTURE 1
   RUNG wire#powerrail
      Contact( "DB2430_FULL_DEPTH".FD_UNIT_02.FIXTURE_2.FD_STA_4_PULSE )
      Contact( "DB8000_PART_STATUS".UNIT_02.FIXTURE_2.PART_A.STATUS.OK )
      I_Contact( "DB8000_PART_STATUS".UNIT_02.FIXTURE_2.PART_A.STATUS.PART_REJECTED )
      wire#w1
      S_Coil( "DB8000_PART_STATUS".UNIT_02.FIXTURE_2.PART_A.STATUS.UNIT_02_STATUS.FACE_N_STATION_4_DONE )
   END_RUNG
   RUNG wire#w1
      R_Coil( "DB8000_PART_STATUS".UNIT_02.FIXTURE_2.PART_A.STATUS.UNIT_02_STATUS.FACE_N_STATION_3_DONE )
   END_RUNG
   // the same network as SCL:
   IF "DB2430_FULL_DEPTH".FD_UNIT_02.FIXTURE_2.FD_STA_4_PULSE AND "DB8000_PART_STATUS".UNIT_02.FIXTURE_2.PART_A.STATUS.OK AND NOT "DB8000_PART_STATUS".UNIT_02.FIXTURE_2.PART_A.STATUS.PART_REJECTED THEN
       "DB8000_PART_STATUS".UNIT_02.FIXTURE_2.PART_A.STATUS.UNIT_02_STATUS.FACE_N_STATION_4_DONE := TRUE;
       "DB8000_PART_STATUS".UNIT_02.FIXTURE_2.PART_A.STATUS.UNIT_02_STATUS.FACE_N_STATION_3_DONE := FALSE;
   END_IF;
END_REGION

REGION Network 23: UNIT 02 FIXTURE 2 TOTAL FULL DEPTH / FULL DEPTH PULSE
   RUNG wire#powerrail
      Contact( "DB2430_FULL_DEPTH".FD_UNIT_02.FIXTURE_2.FULL_DEPTH_STA_1 )
      Contact( "DB2430_FULL_DEPTH".FD_UNIT_02.FIXTURE_2.FULL_DEPTH_STA_2 )
      Contact( "DB2430_FULL_DEPTH".FD_UNIT_02.FIXTURE_2.FULL_DEPTH_STA_3 )
      Contact( "DB2430_FULL_DEPTH".FD_UNIT_02.FIXTURE_2.FULL_DEPTH_STA_4 )
      Contact( "DB7215_PART_TYPE".PART_TYPE_U02_FIXTURES )
      wire#w1
      I_Contact( "DB2430_FULL_DEPTH".FD_UNIT_02.FIXTURE_2.FULL_DEPTH )
      Coil( "DB2430_FULL_DEPTH".FD_UNIT_02.FIXTURE_2.FD_PULSE )
   END_RUNG
   RUNG wire#w1
      Coil( "DB2430_FULL_DEPTH".FD_UNIT_02.FIXTURE_2.FULL_DEPTH )
   END_RUNG
   // the same network as SCL:
   #_w1 := "DB2430_FULL_DEPTH".FD_UNIT_02.FIXTURE_2.FULL_DEPTH_STA_1 AND "DB2430_FULL_DEPTH".FD_UNIT_02.FIXTURE_2.FULL_DEPTH_STA_2 AND "DB2430_FULL_DEPTH".FD_UNIT_02.FIXTURE_2.FULL_DEPTH_STA_3 AND "DB2430_FULL_DEPTH".FD_UNIT_02.FIXTURE_2.FULL_DEPTH_STA_4 AND "DB7215_PART_TYPE".PART_TYPE_U02_FIXTURES;
   "DB2430_FULL_DEPTH".FD_UNIT_02.FIXTURE_2.FD_PULSE := #_w1 AND NOT "DB2430_FULL_DEPTH".FD_UNIT_02.FIXTURE_2.FULL_DEPTH;
   "DB2430_FULL_DEPTH".FD_UNIT_02.FIXTURE_2.FULL_DEPTH := #_w1;
END_REGION

REGION Network 24: UNIT 02 FIXTURE 2 PART TOTAL FULL DEPTH
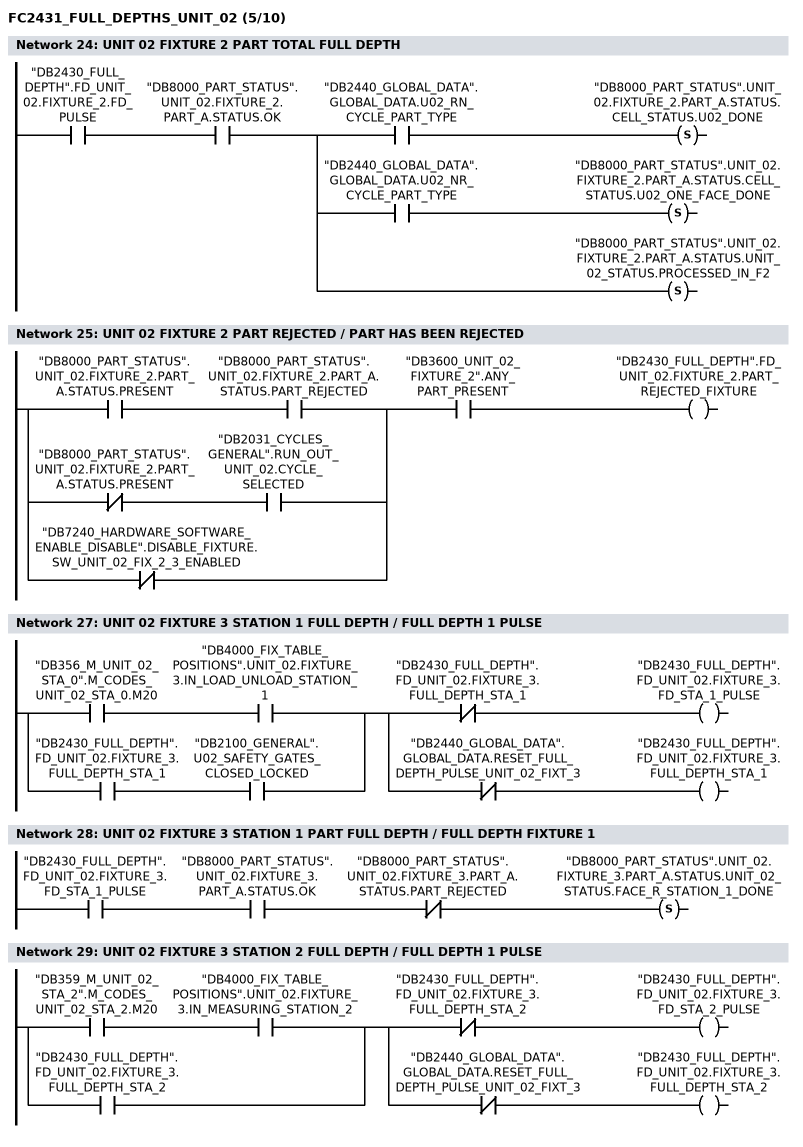
   RUNG wire#powerrail
      Contact( "DB2430_FULL_DEPTH".FD_UNIT_02.FIXTURE_2.FD_PULSE )
      Contact( "DB8000_PART_STATUS".UNIT_02.FIXTURE_2.PART_A.STATUS.OK )
      wire#w1
      Contact( "DB2440_GLOBAL_DATA".GLOBAL_DATA.U02_RN_CYCLE_PART_TYPE )
      S_Coil( "DB8000_PART_STATUS".UNIT_02.FIXTURE_2.PART_A.STATUS.CELL_STATUS.U02_DONE )
   END_RUNG
   RUNG wire#w1
      Contact( "DB2440_GLOBAL_DATA".GLOBAL_DATA.U02_NR_CYCLE_PART_TYPE )
      S_Coil( "DB8000_PART_STATUS".UNIT_02.FIXTURE_2.PART_A.STATUS.CELL_STATUS.U02_ONE_FACE_DONE )
   END_RUNG
   RUNG wire#w1
      S_Coil( "DB8000_PART_STATUS".UNIT_02.FIXTURE_2.PART_A.STATUS.UNIT_02_STATUS.PROCESSED_IN_F2 )
   END_RUNG
   // the same network as SCL:
   #_w1 := "DB2430_FULL_DEPTH".FD_UNIT_02.FIXTURE_2.FD_PULSE AND "DB8000_PART_STATUS".UNIT_02.FIXTURE_2.PART_A.STATUS.OK;
   IF #_w1 AND "DB2440_GLOBAL_DATA".GLOBAL_DATA.U02_RN_CYCLE_PART_TYPE THEN
       "DB8000_PART_STATUS".UNIT_02.FIXTURE_2.PART_A.STATUS.CELL_STATUS.U02_DONE := TRUE;
   END_IF;
   IF #_w1 AND "DB2440_GLOBAL_DATA".GLOBAL_DATA.U02_NR_CYCLE_PART_TYPE THEN
       "DB8000_PART_STATUS".UNIT_02.FIXTURE_2.PART_A.STATUS.CELL_STATUS.U02_ONE_FACE_DONE := TRUE;
   END_IF;
   IF #_w1 THEN
       "DB8000_PART_STATUS".UNIT_02.FIXTURE_2.PART_A.STATUS.UNIT_02_STATUS.PROCESSED_IN_F2 := TRUE;
   END_IF;
END_REGION

REGION Network 25: UNIT 02 FIXTURE 2 PART REJECTED / PART HAS BEEN REJECTED
   RUNG wire#powerrail
      Contact( "DB8000_PART_STATUS".UNIT_02.FIXTURE_2.PART_A.STATUS.PRESENT )
      Contact( "DB8000_PART_STATUS".UNIT_02.FIXTURE_2.PART_A.STATUS.PART_REJECTED )
      wire#w1
      Contact( "DB3600_UNIT_02_FIXTURE_2".ANY_PART_PRESENT )
      Coil( "DB2430_FULL_DEPTH".FD_UNIT_02.FIXTURE_2.PART_REJECTED_FIXTURE )
   END_RUNG
   RUNG wire#powerrail
      I_Contact( "DB8000_PART_STATUS".UNIT_02.FIXTURE_2.PART_A.STATUS.PRESENT )
      Contact( "DB2031_CYCLES_GENERAL".RUN_OUT_UNIT_02.CYCLE_SELECTED )
   END_RUNG wire#w1
   RUNG wire#powerrail
      I_Contact( "DB7240_HARDWARE_SOFTWARE_ENABLE_DISABLE".DISABLE_FIXTURE.SW_UNIT_02_FIX_2_3_ENABLED )
   END_RUNG wire#w1
   // the same network as SCL:
   "DB2430_FULL_DEPTH".FD_UNIT_02.FIXTURE_2.PART_REJECTED_FIXTURE := (("DB8000_PART_STATUS".UNIT_02.FIXTURE_2.PART_A.STATUS.PRESENT AND "DB8000_PART_STATUS".UNIT_02.FIXTURE_2.PART_A.STATUS.PART_REJECTED) OR (NOT "DB8000_PART_STATUS".UNIT_02.FIXTURE_2.PART_A.STATUS.PRESENT AND "DB2031_CYCLES_GENERAL".RUN_OUT_UNIT_02.CYCLE_SELECTED) OR NOT "DB7240_HARDWARE_SOFTWARE_ENABLE_DISABLE".DISABLE_FIXTURE.SW_UNIT_02_FIX_2_3_ENABLED) AND "DB3600_UNIT_02_FIXTURE_2".ANY_PART_PRESENT;
END_REGION

REGION Network 26: <<<<<<<<<<<<<<<<<<<< FIXTURE 3 >>>>>>>>>>>>>>>>>>>>
END_REGION

REGION Network 27: UNIT 02 FIXTURE 3 STATION 1 FULL DEPTH / FULL DEPTH 1 PULSE
   RUNG wire#powerrail
      Contact( "DB356_M_UNIT_02_STA_0".M_CODES_UNIT_02_STA_0.M20 )
      Contact( "DB4000_FIX_TABLE_POSITIONS".UNIT_02.FIXTURE_3.IN_LOAD_UNLOAD_STATION_1 )
      wire#w1
      I_Contact( "DB2430_FULL_DEPTH".FD_UNIT_02.FIXTURE_3.FULL_DEPTH_STA_1 )
      Coil( "DB2430_FULL_DEPTH".FD_UNIT_02.FIXTURE_3.FD_STA_1_PULSE )
   END_RUNG
   RUNG wire#powerrail
      Contact( "DB2430_FULL_DEPTH".FD_UNIT_02.FIXTURE_3.FULL_DEPTH_STA_1 )
      Contact( "DB2100_GENERAL".U02_SAFETY_GATES_CLOSED_LOCKED )
   END_RUNG wire#w1
   RUNG wire#w1
      I_Contact( "DB2440_GLOBAL_DATA".GLOBAL_DATA.RESET_FULL_DEPTH_PULSE_UNIT_02_FIXT_3 )
      Coil( "DB2430_FULL_DEPTH".FD_UNIT_02.FIXTURE_3.FULL_DEPTH_STA_1 )
   END_RUNG
   // the same network as SCL:
   #_w1 := ("DB356_M_UNIT_02_STA_0".M_CODES_UNIT_02_STA_0.M20 AND "DB4000_FIX_TABLE_POSITIONS".UNIT_02.FIXTURE_3.IN_LOAD_UNLOAD_STATION_1) OR ("DB2430_FULL_DEPTH".FD_UNIT_02.FIXTURE_3.FULL_DEPTH_STA_1 AND "DB2100_GENERAL".U02_SAFETY_GATES_CLOSED_LOCKED);
   "DB2430_FULL_DEPTH".FD_UNIT_02.FIXTURE_3.FD_STA_1_PULSE := #_w1 AND NOT "DB2430_FULL_DEPTH".FD_UNIT_02.FIXTURE_3.FULL_DEPTH_STA_1;
   "DB2430_FULL_DEPTH".FD_UNIT_02.FIXTURE_3.FULL_DEPTH_STA_1 := #_w1 AND NOT "DB2440_GLOBAL_DATA".GLOBAL_DATA.RESET_FULL_DEPTH_PULSE_UNIT_02_FIXT_3;
END_REGION

REGION Network 28: UNIT 02 FIXTURE 3 STATION 1 PART FULL DEPTH / FULL DEPTH FIXTURE 1
   RUNG wire#powerrail
      Contact( "DB2430_FULL_DEPTH".FD_UNIT_02.FIXTURE_3.FD_STA_1_PULSE )
      Contact( "DB8000_PART_STATUS".UNIT_02.FIXTURE_3.PART_A.STATUS.OK )
      I_Contact( "DB8000_PART_STATUS".UNIT_02.FIXTURE_3.PART_A.STATUS.PART_REJECTED )
      S_Coil( "DB8000_PART_STATUS".UNIT_02.FIXTURE_3.PART_A.STATUS.UNIT_02_STATUS.FACE_R_STATION_1_DONE )
   END_RUNG
   // the same network as SCL:
   IF "DB2430_FULL_DEPTH".FD_UNIT_02.FIXTURE_3.FD_STA_1_PULSE AND "DB8000_PART_STATUS".UNIT_02.FIXTURE_3.PART_A.STATUS.OK AND NOT "DB8000_PART_STATUS".UNIT_02.FIXTURE_3.PART_A.STATUS.PART_REJECTED THEN
       "DB8000_PART_STATUS".UNIT_02.FIXTURE_3.PART_A.STATUS.UNIT_02_STATUS.FACE_R_STATION_1_DONE := TRUE;
   END_IF;
END_REGION

REGION Network 29: UNIT 02 FIXTURE 3 STATION 2 FULL DEPTH / FULL DEPTH 1 PULSE
   RUNG wire#powerrail
      Contact( "DB359_M_UNIT_02_STA_2".M_CODES_UNIT_02_STA_2.M20 )
      Contact( "DB4000_FIX_TABLE_POSITIONS".UNIT_02.FIXTURE_3.IN_MEASURING_STATION_2 )
      wire#w1
      I_Contact( "DB2430_FULL_DEPTH".FD_UNIT_02.FIXTURE_3.FULL_DEPTH_STA_2 )
      Coil( "DB2430_FULL_DEPTH".FD_UNIT_02.FIXTURE_3.FD_STA_2_PULSE )
   END_RUNG
   RUNG wire#powerrail
      Contact( "DB2430_FULL_DEPTH".FD_UNIT_02.FIXTURE_3.FULL_DEPTH_STA_2 )
   END_RUNG wire#w1
   RUNG wire#w1
      I_Contact( "DB2440_GLOBAL_DATA".GLOBAL_DATA.RESET_FULL_DEPTH_PULSE_UNIT_02_FIXT_3 )
      Coil( "DB2430_FULL_DEPTH".FD_UNIT_02.FIXTURE_3.FULL_DEPTH_STA_2 )
   END_RUNG
   // the same network as SCL:
   #_w1 := ("DB359_M_UNIT_02_STA_2".M_CODES_UNIT_02_STA_2.M20 AND "DB4000_FIX_TABLE_POSITIONS".UNIT_02.FIXTURE_3.IN_MEASURING_STATION_2) OR "DB2430_FULL_DEPTH".FD_UNIT_02.FIXTURE_3.FULL_DEPTH_STA_2;
   "DB2430_FULL_DEPTH".FD_UNIT_02.FIXTURE_3.FD_STA_2_PULSE := #_w1 AND NOT "DB2430_FULL_DEPTH".FD_UNIT_02.FIXTURE_3.FULL_DEPTH_STA_2;
   "DB2430_FULL_DEPTH".FD_UNIT_02.FIXTURE_3.FULL_DEPTH_STA_2 := #_w1 AND NOT "DB2440_GLOBAL_DATA".GLOBAL_DATA.RESET_FULL_DEPTH_PULSE_UNIT_02_FIXT_3;
END_REGION

REGION Network 30: UNIT 02 FIXTURE 3 STATION 2 PART FULL DEPTH / FULL DEPTH FIXTURE 1
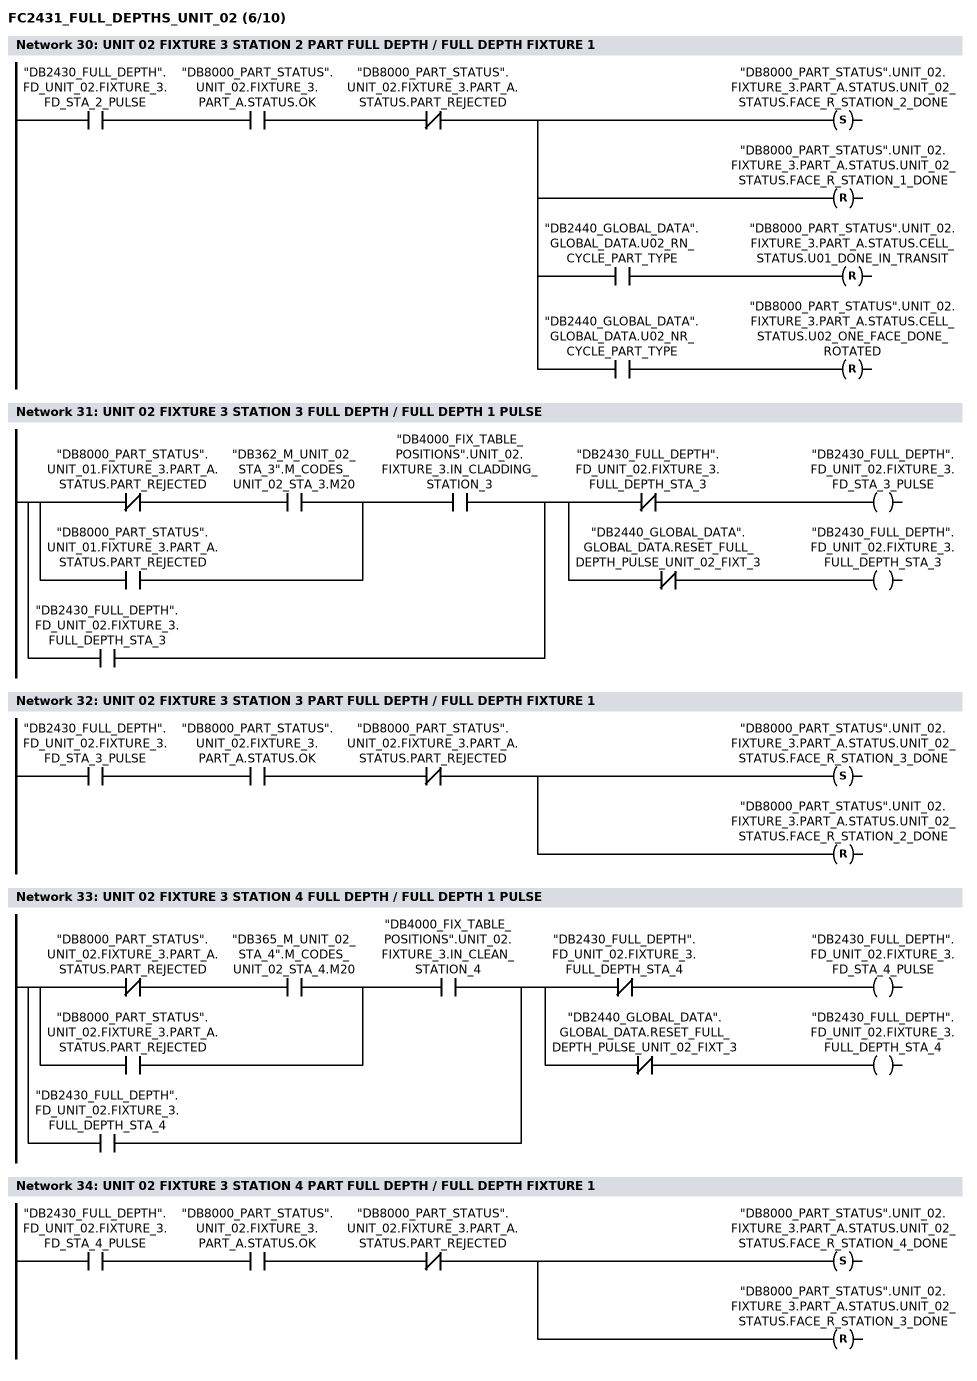
   RUNG wire#powerrail
      Contact( "DB2430_FULL_DEPTH".FD_UNIT_02.FIXTURE_3.FD_STA_2_PULSE )
      Contact( "DB8000_PART_STATUS".UNIT_02.FIXTURE_3.PART_A.STATUS.OK )
      I_Contact( "DB8000_PART_STATUS".UNIT_02.FIXTURE_3.PART_A.STATUS.PART_REJECTED )
      wire#w1
      S_Coil( "DB8000_PART_STATUS".UNIT_02.FIXTURE_3.PART_A.STATUS.UNIT_02_STATUS.FACE_R_STATION_2_DONE )
   END_RUNG
   RUNG wire#w1
      R_Coil( "DB8000_PART_STATUS".UNIT_02.FIXTURE_3.PART_A.STATUS.UNIT_02_STATUS.FACE_R_STATION_1_DONE )
   END_RUNG
   RUNG wire#w1
      Contact( "DB2440_GLOBAL_DATA".GLOBAL_DATA.U02_RN_CYCLE_PART_TYPE )
      R_Coil( "DB8000_PART_STATUS".UNIT_02.FIXTURE_3.PART_A.STATUS.CELL_STATUS.U01_DONE_IN_TRANSIT )
   END_RUNG
   RUNG wire#w1
      Contact( "DB2440_GLOBAL_DATA".GLOBAL_DATA.U02_NR_CYCLE_PART_TYPE )
      R_Coil( "DB8000_PART_STATUS".UNIT_02.FIXTURE_3.PART_A.STATUS.CELL_STATUS.U02_ONE_FACE_DONE_ROTATED )
   END_RUNG
   // the same network as SCL:
   #_w1 := "DB2430_FULL_DEPTH".FD_UNIT_02.FIXTURE_3.FD_STA_2_PULSE AND "DB8000_PART_STATUS".UNIT_02.FIXTURE_3.PART_A.STATUS.OK AND NOT "DB8000_PART_STATUS".UNIT_02.FIXTURE_3.PART_A.STATUS.PART_REJECTED;
   IF #_w1 THEN
       "DB8000_PART_STATUS".UNIT_02.FIXTURE_3.PART_A.STATUS.UNIT_02_STATUS.FACE_R_STATION_2_DONE := TRUE;
       "DB8000_PART_STATUS".UNIT_02.FIXTURE_3.PART_A.STATUS.UNIT_02_STATUS.FACE_R_STATION_1_DONE := FALSE;
   END_IF;
   IF #_w1 AND "DB2440_GLOBAL_DATA".GLOBAL_DATA.U02_RN_CYCLE_PART_TYPE THEN
       "DB8000_PART_STATUS".UNIT_02.FIXTURE_3.PART_A.STATUS.CELL_STATUS.U01_DONE_IN_TRANSIT := FALSE;
   END_IF;
   IF #_w1 AND "DB2440_GLOBAL_DATA".GLOBAL_DATA.U02_NR_CYCLE_PART_TYPE THEN
       "DB8000_PART_STATUS".UNIT_02.FIXTURE_3.PART_A.STATUS.CELL_STATUS.U02_ONE_FACE_DONE_ROTATED := FALSE;
   END_IF;
END_REGION

REGION Network 31: UNIT 02 FIXTURE 3 STATION 3 FULL DEPTH / FULL DEPTH 1 PULSE
   RUNG wire#powerrail
      I_Contact( "DB8000_PART_STATUS".UNIT_01.FIXTURE_3.PART_A.STATUS.PART_REJECTED )
      Contact( "DB362_M_UNIT_02_STA_3".M_CODES_UNIT_02_STA_3.M20 )
      wire#w1
      Contact( "DB4000_FIX_TABLE_POSITIONS".UNIT_02.FIXTURE_3.IN_CLADDING_STATION_3 )
      wire#w2
      I_Contact( "DB2430_FULL_DEPTH".FD_UNIT_02.FIXTURE_3.FULL_DEPTH_STA_3 )
      Coil( "DB2430_FULL_DEPTH".FD_UNIT_02.FIXTURE_3.FD_STA_3_PULSE )
   END_RUNG
   RUNG wire#powerrail
      Contact( "DB8000_PART_STATUS".UNIT_01.FIXTURE_3.PART_A.STATUS.PART_REJECTED )
   END_RUNG wire#w1
   RUNG wire#powerrail
      Contact( "DB2430_FULL_DEPTH".FD_UNIT_02.FIXTURE_3.FULL_DEPTH_STA_3 )
   END_RUNG wire#w2
   RUNG wire#w2
      I_Contact( "DB2440_GLOBAL_DATA".GLOBAL_DATA.RESET_FULL_DEPTH_PULSE_UNIT_02_FIXT_3 )
      Coil( "DB2430_FULL_DEPTH".FD_UNIT_02.FIXTURE_3.FULL_DEPTH_STA_3 )
   END_RUNG
   // the same network as SCL:
   #_w1 := (((NOT "DB8000_PART_STATUS".UNIT_01.FIXTURE_3.PART_A.STATUS.PART_REJECTED AND "DB362_M_UNIT_02_STA_3".M_CODES_UNIT_02_STA_3.M20) OR "DB8000_PART_STATUS".UNIT_01.FIXTURE_3.PART_A.STATUS.PART_REJECTED) AND "DB4000_FIX_TABLE_POSITIONS".UNIT_02.FIXTURE_3.IN_CLADDING_STATION_3) OR "DB2430_FULL_DEPTH".FD_UNIT_02.FIXTURE_3.FULL_DEPTH_STA_3;
   "DB2430_FULL_DEPTH".FD_UNIT_02.FIXTURE_3.FD_STA_3_PULSE := #_w1 AND NOT "DB2430_FULL_DEPTH".FD_UNIT_02.FIXTURE_3.FULL_DEPTH_STA_3;
   "DB2430_FULL_DEPTH".FD_UNIT_02.FIXTURE_3.FULL_DEPTH_STA_3 := #_w1 AND NOT "DB2440_GLOBAL_DATA".GLOBAL_DATA.RESET_FULL_DEPTH_PULSE_UNIT_02_FIXT_3;
END_REGION

REGION Network 32: UNIT 02 FIXTURE 3 STATION 3 PART FULL DEPTH / FULL DEPTH FIXTURE 1
   RUNG wire#powerrail
      Contact( "DB2430_FULL_DEPTH".FD_UNIT_02.FIXTURE_3.FD_STA_3_PULSE )
      Contact( "DB8000_PART_STATUS".UNIT_02.FIXTURE_3.PART_A.STATUS.OK )
      I_Contact( "DB8000_PART_STATUS".UNIT_02.FIXTURE_3.PART_A.STATUS.PART_REJECTED )
      wire#w1
      S_Coil( "DB8000_PART_STATUS".UNIT_02.FIXTURE_3.PART_A.STATUS.UNIT_02_STATUS.FACE_R_STATION_3_DONE )
   END_RUNG
   RUNG wire#w1
      R_Coil( "DB8000_PART_STATUS".UNIT_02.FIXTURE_3.PART_A.STATUS.UNIT_02_STATUS.FACE_R_STATION_2_DONE )
   END_RUNG
   // the same network as SCL:
   IF "DB2430_FULL_DEPTH".FD_UNIT_02.FIXTURE_3.FD_STA_3_PULSE AND "DB8000_PART_STATUS".UNIT_02.FIXTURE_3.PART_A.STATUS.OK AND NOT "DB8000_PART_STATUS".UNIT_02.FIXTURE_3.PART_A.STATUS.PART_REJECTED THEN
       "DB8000_PART_STATUS".UNIT_02.FIXTURE_3.PART_A.STATUS.UNIT_02_STATUS.FACE_R_STATION_3_DONE := TRUE;
       "DB8000_PART_STATUS".UNIT_02.FIXTURE_3.PART_A.STATUS.UNIT_02_STATUS.FACE_R_STATION_2_DONE := FALSE;
   END_IF;
END_REGION

REGION Network 33: UNIT 02 FIXTURE 3 STATION 4 FULL DEPTH / FULL DEPTH 1 PULSE
   RUNG wire#powerrail
      I_Contact( "DB8000_PART_STATUS".UNIT_02.FIXTURE_3.PART_A.STATUS.PART_REJECTED )
      Contact( "DB365_M_UNIT_02_STA_4".M_CODES_UNIT_02_STA_4.M20 )
      wire#w1
      Contact( "DB4000_FIX_TABLE_POSITIONS".UNIT_02.FIXTURE_3.IN_CLEAN_STATION_4 )
      wire#w2
      I_Contact( "DB2430_FULL_DEPTH".FD_UNIT_02.FIXTURE_3.FULL_DEPTH_STA_4 )
      Coil( "DB2430_FULL_DEPTH".FD_UNIT_02.FIXTURE_3.FD_STA_4_PULSE )
   END_RUNG
   RUNG wire#powerrail
      Contact( "DB8000_PART_STATUS".UNIT_02.FIXTURE_3.PART_A.STATUS.PART_REJECTED )
   END_RUNG wire#w1
   RUNG wire#powerrail
      Contact( "DB2430_FULL_DEPTH".FD_UNIT_02.FIXTURE_3.FULL_DEPTH_STA_4 )
   END_RUNG wire#w2
   RUNG wire#w2
      I_Contact( "DB2440_GLOBAL_DATA".GLOBAL_DATA.RESET_FULL_DEPTH_PULSE_UNIT_02_FIXT_3 )
      Coil( "DB2430_FULL_DEPTH".FD_UNIT_02.FIXTURE_3.FULL_DEPTH_STA_4 )
   END_RUNG
   // the same network as SCL:
   #_w1 := (((NOT "DB8000_PART_STATUS".UNIT_02.FIXTURE_3.PART_A.STATUS.PART_REJECTED AND "DB365_M_UNIT_02_STA_4".M_CODES_UNIT_02_STA_4.M20) OR "DB8000_PART_STATUS".UNIT_02.FIXTURE_3.PART_A.STATUS.PART_REJECTED) AND "DB4000_FIX_TABLE_POSITIONS".UNIT_02.FIXTURE_3.IN_CLEAN_STATION_4) OR "DB2430_FULL_DEPTH".FD_UNIT_02.FIXTURE_3.FULL_DEPTH_STA_4;
   "DB2430_FULL_DEPTH".FD_UNIT_02.FIXTURE_3.FD_STA_4_PULSE := #_w1 AND NOT "DB2430_FULL_DEPTH".FD_UNIT_02.FIXTURE_3.FULL_DEPTH_STA_4;
   "DB2430_FULL_DEPTH".FD_UNIT_02.FIXTURE_3.FULL_DEPTH_STA_4 := #_w1 AND NOT "DB2440_GLOBAL_DATA".GLOBAL_DATA.RESET_FULL_DEPTH_PULSE_UNIT_02_FIXT_3;
END_REGION

REGION Network 34: UNIT 02 FIXTURE 3 STATION 4 PART FULL DEPTH / FULL DEPTH FIXTURE 1
   RUNG wire#powerrail
      Contact( "DB2430_FULL_DEPTH".FD_UNIT_02.FIXTURE_3.FD_STA_4_PULSE )
      Contact( "DB8000_PART_STATUS".UNIT_02.FIXTURE_3.PART_A.STATUS.OK )
      I_Contact( "DB8000_PART_STATUS".UNIT_02.FIXTURE_3.PART_A.STATUS.PART_REJECTED )
      wire#w1
      S_Coil( "DB8000_PART_STATUS".UNIT_02.FIXTURE_3.PART_A.STATUS.UNIT_02_STATUS.FACE_R_STATION_4_DONE )
   END_RUNG
   RUNG wire#w1
      R_Coil( "DB8000_PART_STATUS".UNIT_02.FIXTURE_3.PART_A.STATUS.UNIT_02_STATUS.FACE_R_STATION_3_DONE )
   END_RUNG
   // the same network as SCL:
   IF "DB2430_FULL_DEPTH".FD_UNIT_02.FIXTURE_3.FD_STA_4_PULSE AND "DB8000_PART_STATUS".UNIT_02.FIXTURE_3.PART_A.STATUS.OK AND NOT "DB8000_PART_STATUS".UNIT_02.FIXTURE_3.PART_A.STATUS.PART_REJECTED THEN
       "DB8000_PART_STATUS".UNIT_02.FIXTURE_3.PART_A.STATUS.UNIT_02_STATUS.FACE_R_STATION_4_DONE := TRUE;
       "DB8000_PART_STATUS".UNIT_02.FIXTURE_3.PART_A.STATUS.UNIT_02_STATUS.FACE_R_STATION_3_DONE := FALSE;
   END_IF;
END_REGION

REGION Network 35: UNIT 02 FIXTURE 3 TOTAL FULL DEPTH / FULL DEPTH PULSE
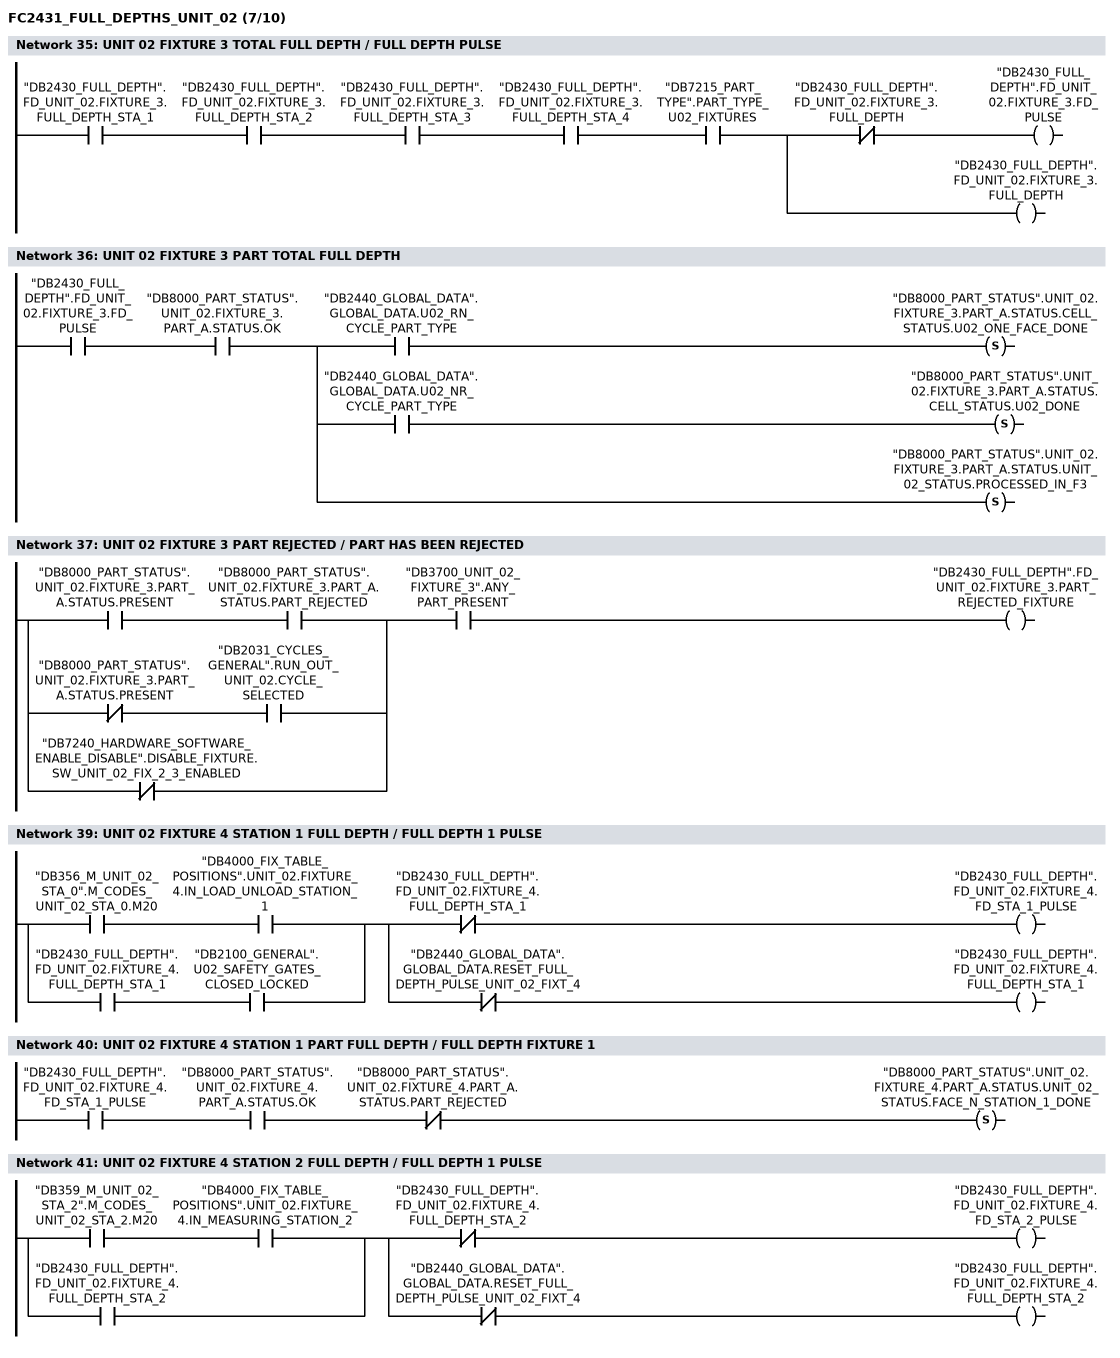
   RUNG wire#powerrail
      Contact( "DB2430_FULL_DEPTH".FD_UNIT_02.FIXTURE_3.FULL_DEPTH_STA_1 )
      Contact( "DB2430_FULL_DEPTH".FD_UNIT_02.FIXTURE_3.FULL_DEPTH_STA_2 )
      Contact( "DB2430_FULL_DEPTH".FD_UNIT_02.FIXTURE_3.FULL_DEPTH_STA_3 )
      Contact( "DB2430_FULL_DEPTH".FD_UNIT_02.FIXTURE_3.FULL_DEPTH_STA_4 )
      Contact( "DB7215_PART_TYPE".PART_TYPE_U02_FIXTURES )
      wire#w1
      I_Contact( "DB2430_FULL_DEPTH".FD_UNIT_02.FIXTURE_3.FULL_DEPTH )
      Coil( "DB2430_FULL_DEPTH".FD_UNIT_02.FIXTURE_3.FD_PULSE )
   END_RUNG
   RUNG wire#w1
      Coil( "DB2430_FULL_DEPTH".FD_UNIT_02.FIXTURE_3.FULL_DEPTH )
   END_RUNG
   // the same network as SCL:
   #_w1 := "DB2430_FULL_DEPTH".FD_UNIT_02.FIXTURE_3.FULL_DEPTH_STA_1 AND "DB2430_FULL_DEPTH".FD_UNIT_02.FIXTURE_3.FULL_DEPTH_STA_2 AND "DB2430_FULL_DEPTH".FD_UNIT_02.FIXTURE_3.FULL_DEPTH_STA_3 AND "DB2430_FULL_DEPTH".FD_UNIT_02.FIXTURE_3.FULL_DEPTH_STA_4 AND "DB7215_PART_TYPE".PART_TYPE_U02_FIXTURES;
   "DB2430_FULL_DEPTH".FD_UNIT_02.FIXTURE_3.FD_PULSE := #_w1 AND NOT "DB2430_FULL_DEPTH".FD_UNIT_02.FIXTURE_3.FULL_DEPTH;
   "DB2430_FULL_DEPTH".FD_UNIT_02.FIXTURE_3.FULL_DEPTH := #_w1;
END_REGION

REGION Network 36: UNIT 02 FIXTURE 3 PART TOTAL FULL DEPTH
   RUNG wire#powerrail
      Contact( "DB2430_FULL_DEPTH".FD_UNIT_02.FIXTURE_3.FD_PULSE )
      Contact( "DB8000_PART_STATUS".UNIT_02.FIXTURE_3.PART_A.STATUS.OK )
      wire#w1
      Contact( "DB2440_GLOBAL_DATA".GLOBAL_DATA.U02_RN_CYCLE_PART_TYPE )
      S_Coil( "DB8000_PART_STATUS".UNIT_02.FIXTURE_3.PART_A.STATUS.CELL_STATUS.U02_ONE_FACE_DONE )
   END_RUNG
   RUNG wire#w1
      Contact( "DB2440_GLOBAL_DATA".GLOBAL_DATA.U02_NR_CYCLE_PART_TYPE )
      S_Coil( "DB8000_PART_STATUS".UNIT_02.FIXTURE_3.PART_A.STATUS.CELL_STATUS.U02_DONE )
   END_RUNG
   RUNG wire#w1
      S_Coil( "DB8000_PART_STATUS".UNIT_02.FIXTURE_3.PART_A.STATUS.UNIT_02_STATUS.PROCESSED_IN_F3 )
   END_RUNG
   // the same network as SCL:
   #_w1 := "DB2430_FULL_DEPTH".FD_UNIT_02.FIXTURE_3.FD_PULSE AND "DB8000_PART_STATUS".UNIT_02.FIXTURE_3.PART_A.STATUS.OK;
   IF #_w1 AND "DB2440_GLOBAL_DATA".GLOBAL_DATA.U02_RN_CYCLE_PART_TYPE THEN
       "DB8000_PART_STATUS".UNIT_02.FIXTURE_3.PART_A.STATUS.CELL_STATUS.U02_ONE_FACE_DONE := TRUE;
   END_IF;
   IF #_w1 AND "DB2440_GLOBAL_DATA".GLOBAL_DATA.U02_NR_CYCLE_PART_TYPE THEN
       "DB8000_PART_STATUS".UNIT_02.FIXTURE_3.PART_A.STATUS.CELL_STATUS.U02_DONE := TRUE;
   END_IF;
   IF #_w1 THEN
       "DB8000_PART_STATUS".UNIT_02.FIXTURE_3.PART_A.STATUS.UNIT_02_STATUS.PROCESSED_IN_F3 := TRUE;
   END_IF;
END_REGION

REGION Network 37: UNIT 02 FIXTURE 3 PART REJECTED / PART HAS BEEN REJECTED
   RUNG wire#powerrail
      Contact( "DB8000_PART_STATUS".UNIT_02.FIXTURE_3.PART_A.STATUS.PRESENT )
      Contact( "DB8000_PART_STATUS".UNIT_02.FIXTURE_3.PART_A.STATUS.PART_REJECTED )
      wire#w1
      Contact( "DB3700_UNIT_02_FIXTURE_3".ANY_PART_PRESENT )
      Coil( "DB2430_FULL_DEPTH".FD_UNIT_02.FIXTURE_3.PART_REJECTED_FIXTURE )
   END_RUNG
   RUNG wire#powerrail
      I_Contact( "DB8000_PART_STATUS".UNIT_02.FIXTURE_3.PART_A.STATUS.PRESENT )
      Contact( "DB2031_CYCLES_GENERAL".RUN_OUT_UNIT_02.CYCLE_SELECTED )
   END_RUNG wire#w1
   RUNG wire#powerrail
      I_Contact( "DB7240_HARDWARE_SOFTWARE_ENABLE_DISABLE".DISABLE_FIXTURE.SW_UNIT_02_FIX_2_3_ENABLED )
   END_RUNG wire#w1
   // the same network as SCL:
   "DB2430_FULL_DEPTH".FD_UNIT_02.FIXTURE_3.PART_REJECTED_FIXTURE := (("DB8000_PART_STATUS".UNIT_02.FIXTURE_3.PART_A.STATUS.PRESENT AND "DB8000_PART_STATUS".UNIT_02.FIXTURE_3.PART_A.STATUS.PART_REJECTED) OR (NOT "DB8000_PART_STATUS".UNIT_02.FIXTURE_3.PART_A.STATUS.PRESENT AND "DB2031_CYCLES_GENERAL".RUN_OUT_UNIT_02.CYCLE_SELECTED) OR NOT "DB7240_HARDWARE_SOFTWARE_ENABLE_DISABLE".DISABLE_FIXTURE.SW_UNIT_02_FIX_2_3_ENABLED) AND "DB3700_UNIT_02_FIXTURE_3".ANY_PART_PRESENT;
END_REGION

REGION Network 38: <<<<<<<<<<<<<<<<<<<< FIXTURE 4 >>>>>>>>>>>>>>>>>>>>
END_REGION

REGION Network 39: UNIT 02 FIXTURE 4 STATION 1 FULL DEPTH / FULL DEPTH 1 PULSE
   RUNG wire#powerrail
      Contact( "DB356_M_UNIT_02_STA_0".M_CODES_UNIT_02_STA_0.M20 )
      Contact( "DB4000_FIX_TABLE_POSITIONS".UNIT_02.FIXTURE_4.IN_LOAD_UNLOAD_STATION_1 )
      wire#w1
      I_Contact( "DB2430_FULL_DEPTH".FD_UNIT_02.FIXTURE_4.FULL_DEPTH_STA_1 )
      Coil( "DB2430_FULL_DEPTH".FD_UNIT_02.FIXTURE_4.FD_STA_1_PULSE )
   END_RUNG
   RUNG wire#powerrail
      Contact( "DB2430_FULL_DEPTH".FD_UNIT_02.FIXTURE_4.FULL_DEPTH_STA_1 )
      Contact( "DB2100_GENERAL".U02_SAFETY_GATES_CLOSED_LOCKED )
   END_RUNG wire#w1
   RUNG wire#w1
      I_Contact( "DB2440_GLOBAL_DATA".GLOBAL_DATA.RESET_FULL_DEPTH_PULSE_UNIT_02_FIXT_4 )
      Coil( "DB2430_FULL_DEPTH".FD_UNIT_02.FIXTURE_4.FULL_DEPTH_STA_1 )
   END_RUNG
   // the same network as SCL:
   #_w1 := ("DB356_M_UNIT_02_STA_0".M_CODES_UNIT_02_STA_0.M20 AND "DB4000_FIX_TABLE_POSITIONS".UNIT_02.FIXTURE_4.IN_LOAD_UNLOAD_STATION_1) OR ("DB2430_FULL_DEPTH".FD_UNIT_02.FIXTURE_4.FULL_DEPTH_STA_1 AND "DB2100_GENERAL".U02_SAFETY_GATES_CLOSED_LOCKED);
   "DB2430_FULL_DEPTH".FD_UNIT_02.FIXTURE_4.FD_STA_1_PULSE := #_w1 AND NOT "DB2430_FULL_DEPTH".FD_UNIT_02.FIXTURE_4.FULL_DEPTH_STA_1;
   "DB2430_FULL_DEPTH".FD_UNIT_02.FIXTURE_4.FULL_DEPTH_STA_1 := #_w1 AND NOT "DB2440_GLOBAL_DATA".GLOBAL_DATA.RESET_FULL_DEPTH_PULSE_UNIT_02_FIXT_4;
END_REGION

REGION Network 40: UNIT 02 FIXTURE 4 STATION 1 PART FULL DEPTH / FULL DEPTH FIXTURE 1
   RUNG wire#powerrail
      Contact( "DB2430_FULL_DEPTH".FD_UNIT_02.FIXTURE_4.FD_STA_1_PULSE )
      Contact( "DB8000_PART_STATUS".UNIT_02.FIXTURE_4.PART_A.STATUS.OK )
      I_Contact( "DB8000_PART_STATUS".UNIT_02.FIXTURE_4.PART_A.STATUS.PART_REJECTED )
      S_Coil( "DB8000_PART_STATUS".UNIT_02.FIXTURE_4.PART_A.STATUS.UNIT_02_STATUS.FACE_N_STATION_1_DONE )
   END_RUNG
   // the same network as SCL:
   IF "DB2430_FULL_DEPTH".FD_UNIT_02.FIXTURE_4.FD_STA_1_PULSE AND "DB8000_PART_STATUS".UNIT_02.FIXTURE_4.PART_A.STATUS.OK AND NOT "DB8000_PART_STATUS".UNIT_02.FIXTURE_4.PART_A.STATUS.PART_REJECTED THEN
       "DB8000_PART_STATUS".UNIT_02.FIXTURE_4.PART_A.STATUS.UNIT_02_STATUS.FACE_N_STATION_1_DONE := TRUE;
   END_IF;
END_REGION

REGION Network 41: UNIT 02 FIXTURE 4 STATION 2 FULL DEPTH / FULL DEPTH 1 PULSE
   RUNG wire#powerrail
      Contact( "DB359_M_UNIT_02_STA_2".M_CODES_UNIT_02_STA_2.M20 )
      Contact( "DB4000_FIX_TABLE_POSITIONS".UNIT_02.FIXTURE_4.IN_MEASURING_STATION_2 )
      wire#w1
      I_Contact( "DB2430_FULL_DEPTH".FD_UNIT_02.FIXTURE_4.FULL_DEPTH_STA_2 )
      Coil( "DB2430_FULL_DEPTH".FD_UNIT_02.FIXTURE_4.FD_STA_2_PULSE )
   END_RUNG
   RUNG wire#powerrail
      Contact( "DB2430_FULL_DEPTH".FD_UNIT_02.FIXTURE_4.FULL_DEPTH_STA_2 )
   END_RUNG wire#w1
   RUNG wire#w1
      I_Contact( "DB2440_GLOBAL_DATA".GLOBAL_DATA.RESET_FULL_DEPTH_PULSE_UNIT_02_FIXT_4 )
      Coil( "DB2430_FULL_DEPTH".FD_UNIT_02.FIXTURE_4.FULL_DEPTH_STA_2 )
   END_RUNG
   // the same network as SCL:
   #_w1 := ("DB359_M_UNIT_02_STA_2".M_CODES_UNIT_02_STA_2.M20 AND "DB4000_FIX_TABLE_POSITIONS".UNIT_02.FIXTURE_4.IN_MEASURING_STATION_2) OR "DB2430_FULL_DEPTH".FD_UNIT_02.FIXTURE_4.FULL_DEPTH_STA_2;
   "DB2430_FULL_DEPTH".FD_UNIT_02.FIXTURE_4.FD_STA_2_PULSE := #_w1 AND NOT "DB2430_FULL_DEPTH".FD_UNIT_02.FIXTURE_4.FULL_DEPTH_STA_2;
   "DB2430_FULL_DEPTH".FD_UNIT_02.FIXTURE_4.FULL_DEPTH_STA_2 := #_w1 AND NOT "DB2440_GLOBAL_DATA".GLOBAL_DATA.RESET_FULL_DEPTH_PULSE_UNIT_02_FIXT_4;
END_REGION

REGION Network 42: UNIT 02 FIXTURE 4 STATION 2 PART FULL DEPTH / FULL DEPTH FIXTURE 1
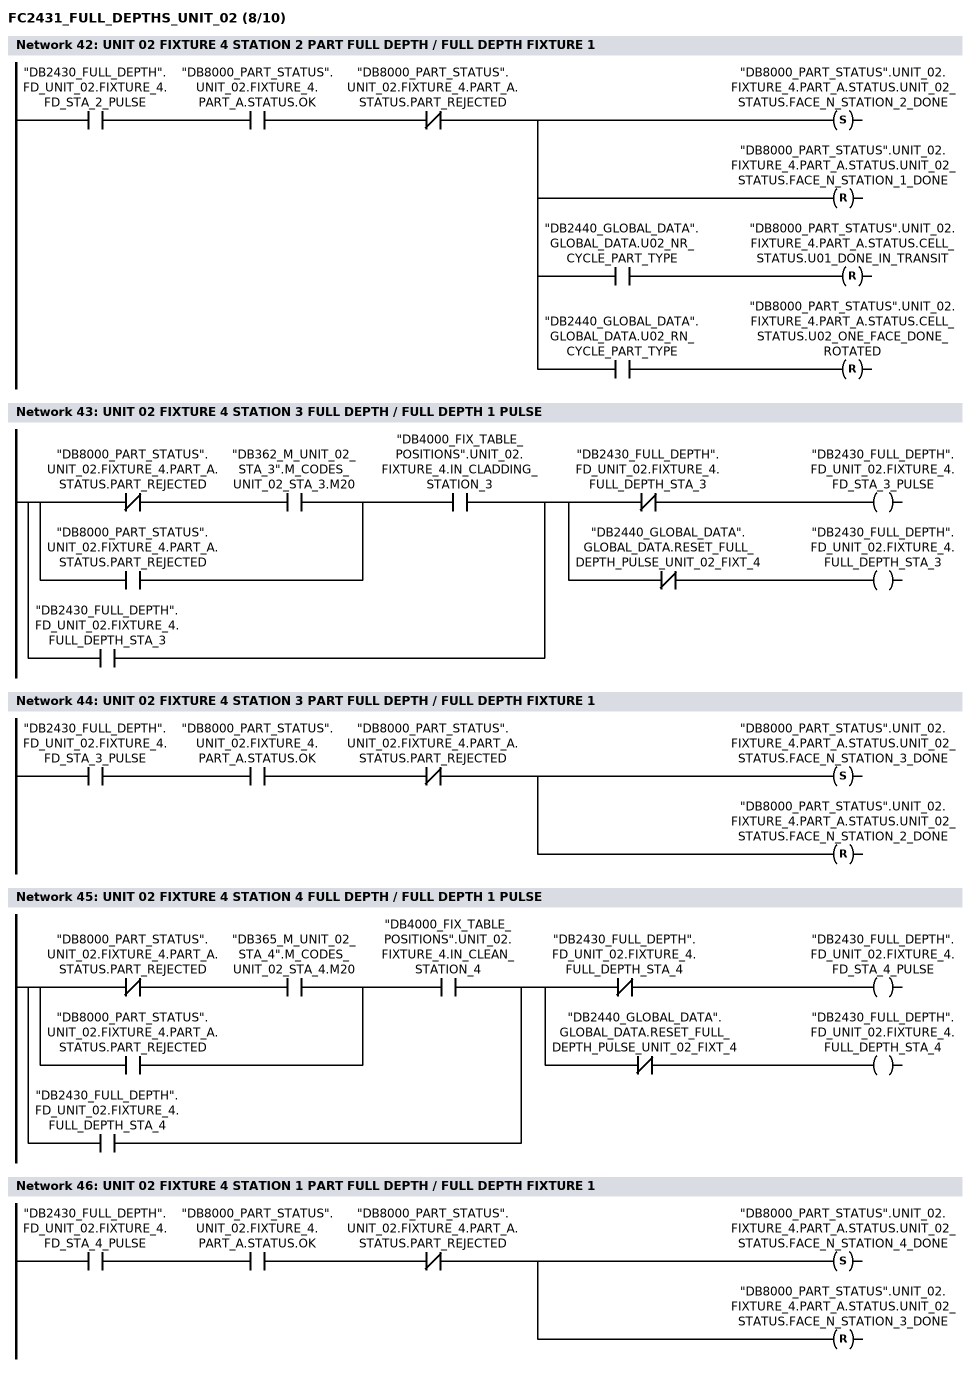
   RUNG wire#powerrail
      Contact( "DB2430_FULL_DEPTH".FD_UNIT_02.FIXTURE_4.FD_STA_2_PULSE )
      Contact( "DB8000_PART_STATUS".UNIT_02.FIXTURE_4.PART_A.STATUS.OK )
      I_Contact( "DB8000_PART_STATUS".UNIT_02.FIXTURE_4.PART_A.STATUS.PART_REJECTED )
      wire#w1
      S_Coil( "DB8000_PART_STATUS".UNIT_02.FIXTURE_4.PART_A.STATUS.UNIT_02_STATUS.FACE_N_STATION_2_DONE )
   END_RUNG
   RUNG wire#w1
      R_Coil( "DB8000_PART_STATUS".UNIT_02.FIXTURE_4.PART_A.STATUS.UNIT_02_STATUS.FACE_N_STATION_1_DONE )
   END_RUNG
   RUNG wire#w1
      Contact( "DB2440_GLOBAL_DATA".GLOBAL_DATA.U02_NR_CYCLE_PART_TYPE )
      R_Coil( "DB8000_PART_STATUS".UNIT_02.FIXTURE_4.PART_A.STATUS.CELL_STATUS.U01_DONE_IN_TRANSIT )
   END_RUNG
   RUNG wire#w1
      Contact( "DB2440_GLOBAL_DATA".GLOBAL_DATA.U02_RN_CYCLE_PART_TYPE )
      R_Coil( "DB8000_PART_STATUS".UNIT_02.FIXTURE_4.PART_A.STATUS.CELL_STATUS.U02_ONE_FACE_DONE_ROTATED )
   END_RUNG
   // the same network as SCL:
   #_w1 := "DB2430_FULL_DEPTH".FD_UNIT_02.FIXTURE_4.FD_STA_2_PULSE AND "DB8000_PART_STATUS".UNIT_02.FIXTURE_4.PART_A.STATUS.OK AND NOT "DB8000_PART_STATUS".UNIT_02.FIXTURE_4.PART_A.STATUS.PART_REJECTED;
   IF #_w1 THEN
       "DB8000_PART_STATUS".UNIT_02.FIXTURE_4.PART_A.STATUS.UNIT_02_STATUS.FACE_N_STATION_2_DONE := TRUE;
       "DB8000_PART_STATUS".UNIT_02.FIXTURE_4.PART_A.STATUS.UNIT_02_STATUS.FACE_N_STATION_1_DONE := FALSE;
   END_IF;
   IF #_w1 AND "DB2440_GLOBAL_DATA".GLOBAL_DATA.U02_NR_CYCLE_PART_TYPE THEN
       "DB8000_PART_STATUS".UNIT_02.FIXTURE_4.PART_A.STATUS.CELL_STATUS.U01_DONE_IN_TRANSIT := FALSE;
   END_IF;
   IF #_w1 AND "DB2440_GLOBAL_DATA".GLOBAL_DATA.U02_RN_CYCLE_PART_TYPE THEN
       "DB8000_PART_STATUS".UNIT_02.FIXTURE_4.PART_A.STATUS.CELL_STATUS.U02_ONE_FACE_DONE_ROTATED := FALSE;
   END_IF;
END_REGION

REGION Network 43: UNIT 02 FIXTURE 4 STATION 3 FULL DEPTH / FULL DEPTH 1 PULSE
   RUNG wire#powerrail
      I_Contact( "DB8000_PART_STATUS".UNIT_02.FIXTURE_4.PART_A.STATUS.PART_REJECTED )
      Contact( "DB362_M_UNIT_02_STA_3".M_CODES_UNIT_02_STA_3.M20 )
      wire#w1
      Contact( "DB4000_FIX_TABLE_POSITIONS".UNIT_02.FIXTURE_4.IN_CLADDING_STATION_3 )
      wire#w2
      I_Contact( "DB2430_FULL_DEPTH".FD_UNIT_02.FIXTURE_4.FULL_DEPTH_STA_3 )
      Coil( "DB2430_FULL_DEPTH".FD_UNIT_02.FIXTURE_4.FD_STA_3_PULSE )
   END_RUNG
   RUNG wire#powerrail
      Contact( "DB8000_PART_STATUS".UNIT_02.FIXTURE_4.PART_A.STATUS.PART_REJECTED )
   END_RUNG wire#w1
   RUNG wire#powerrail
      Contact( "DB2430_FULL_DEPTH".FD_UNIT_02.FIXTURE_4.FULL_DEPTH_STA_3 )
   END_RUNG wire#w2
   RUNG wire#w2
      I_Contact( "DB2440_GLOBAL_DATA".GLOBAL_DATA.RESET_FULL_DEPTH_PULSE_UNIT_02_FIXT_4 )
      Coil( "DB2430_FULL_DEPTH".FD_UNIT_02.FIXTURE_4.FULL_DEPTH_STA_3 )
   END_RUNG
   // the same network as SCL:
   #_w1 := (((NOT "DB8000_PART_STATUS".UNIT_02.FIXTURE_4.PART_A.STATUS.PART_REJECTED AND "DB362_M_UNIT_02_STA_3".M_CODES_UNIT_02_STA_3.M20) OR "DB8000_PART_STATUS".UNIT_02.FIXTURE_4.PART_A.STATUS.PART_REJECTED) AND "DB4000_FIX_TABLE_POSITIONS".UNIT_02.FIXTURE_4.IN_CLADDING_STATION_3) OR "DB2430_FULL_DEPTH".FD_UNIT_02.FIXTURE_4.FULL_DEPTH_STA_3;
   "DB2430_FULL_DEPTH".FD_UNIT_02.FIXTURE_4.FD_STA_3_PULSE := #_w1 AND NOT "DB2430_FULL_DEPTH".FD_UNIT_02.FIXTURE_4.FULL_DEPTH_STA_3;
   "DB2430_FULL_DEPTH".FD_UNIT_02.FIXTURE_4.FULL_DEPTH_STA_3 := #_w1 AND NOT "DB2440_GLOBAL_DATA".GLOBAL_DATA.RESET_FULL_DEPTH_PULSE_UNIT_02_FIXT_4;
END_REGION

REGION Network 44: UNIT 02 FIXTURE 4 STATION 3 PART FULL DEPTH / FULL DEPTH FIXTURE 1
   RUNG wire#powerrail
      Contact( "DB2430_FULL_DEPTH".FD_UNIT_02.FIXTURE_4.FD_STA_3_PULSE )
      Contact( "DB8000_PART_STATUS".UNIT_02.FIXTURE_4.PART_A.STATUS.OK )
      I_Contact( "DB8000_PART_STATUS".UNIT_02.FIXTURE_4.PART_A.STATUS.PART_REJECTED )
      wire#w1
      S_Coil( "DB8000_PART_STATUS".UNIT_02.FIXTURE_4.PART_A.STATUS.UNIT_02_STATUS.FACE_N_STATION_3_DONE )
   END_RUNG
   RUNG wire#w1
      R_Coil( "DB8000_PART_STATUS".UNIT_02.FIXTURE_4.PART_A.STATUS.UNIT_02_STATUS.FACE_N_STATION_2_DONE )
   END_RUNG
   // the same network as SCL:
   IF "DB2430_FULL_DEPTH".FD_UNIT_02.FIXTURE_4.FD_STA_3_PULSE AND "DB8000_PART_STATUS".UNIT_02.FIXTURE_4.PART_A.STATUS.OK AND NOT "DB8000_PART_STATUS".UNIT_02.FIXTURE_4.PART_A.STATUS.PART_REJECTED THEN
       "DB8000_PART_STATUS".UNIT_02.FIXTURE_4.PART_A.STATUS.UNIT_02_STATUS.FACE_N_STATION_3_DONE := TRUE;
       "DB8000_PART_STATUS".UNIT_02.FIXTURE_4.PART_A.STATUS.UNIT_02_STATUS.FACE_N_STATION_2_DONE := FALSE;
   END_IF;
END_REGION

REGION Network 45: UNIT 02 FIXTURE 4 STATION 4 FULL DEPTH / FULL DEPTH 1 PULSE
   RUNG wire#powerrail
      I_Contact( "DB8000_PART_STATUS".UNIT_02.FIXTURE_4.PART_A.STATUS.PART_REJECTED )
      Contact( "DB365_M_UNIT_02_STA_4".M_CODES_UNIT_02_STA_4.M20 )
      wire#w1
      Contact( "DB4000_FIX_TABLE_POSITIONS".UNIT_02.FIXTURE_4.IN_CLEAN_STATION_4 )
      wire#w2
      I_Contact( "DB2430_FULL_DEPTH".FD_UNIT_02.FIXTURE_4.FULL_DEPTH_STA_4 )
      Coil( "DB2430_FULL_DEPTH".FD_UNIT_02.FIXTURE_4.FD_STA_4_PULSE )
   END_RUNG
   RUNG wire#powerrail
      Contact( "DB8000_PART_STATUS".UNIT_02.FIXTURE_4.PART_A.STATUS.PART_REJECTED )
   END_RUNG wire#w1
   RUNG wire#powerrail
      Contact( "DB2430_FULL_DEPTH".FD_UNIT_02.FIXTURE_4.FULL_DEPTH_STA_4 )
   END_RUNG wire#w2
   RUNG wire#w2
      I_Contact( "DB2440_GLOBAL_DATA".GLOBAL_DATA.RESET_FULL_DEPTH_PULSE_UNIT_02_FIXT_4 )
      Coil( "DB2430_FULL_DEPTH".FD_UNIT_02.FIXTURE_4.FULL_DEPTH_STA_4 )
   END_RUNG
   // the same network as SCL:
   #_w1 := (((NOT "DB8000_PART_STATUS".UNIT_02.FIXTURE_4.PART_A.STATUS.PART_REJECTED AND "DB365_M_UNIT_02_STA_4".M_CODES_UNIT_02_STA_4.M20) OR "DB8000_PART_STATUS".UNIT_02.FIXTURE_4.PART_A.STATUS.PART_REJECTED) AND "DB4000_FIX_TABLE_POSITIONS".UNIT_02.FIXTURE_4.IN_CLEAN_STATION_4) OR "DB2430_FULL_DEPTH".FD_UNIT_02.FIXTURE_4.FULL_DEPTH_STA_4;
   "DB2430_FULL_DEPTH".FD_UNIT_02.FIXTURE_4.FD_STA_4_PULSE := #_w1 AND NOT "DB2430_FULL_DEPTH".FD_UNIT_02.FIXTURE_4.FULL_DEPTH_STA_4;
   "DB2430_FULL_DEPTH".FD_UNIT_02.FIXTURE_4.FULL_DEPTH_STA_4 := #_w1 AND NOT "DB2440_GLOBAL_DATA".GLOBAL_DATA.RESET_FULL_DEPTH_PULSE_UNIT_02_FIXT_4;
END_REGION

REGION Network 46: UNIT 02 FIXTURE 4 STATION 1 PART FULL DEPTH / FULL DEPTH FIXTURE 1
   RUNG wire#powerrail
      Contact( "DB2430_FULL_DEPTH".FD_UNIT_02.FIXTURE_4.FD_STA_4_PULSE )
      Contact( "DB8000_PART_STATUS".UNIT_02.FIXTURE_4.PART_A.STATUS.OK )
      I_Contact( "DB8000_PART_STATUS".UNIT_02.FIXTURE_4.PART_A.STATUS.PART_REJECTED )
      wire#w1
      S_Coil( "DB8000_PART_STATUS".UNIT_02.FIXTURE_4.PART_A.STATUS.UNIT_02_STATUS.FACE_N_STATION_4_DONE )
   END_RUNG
   RUNG wire#w1
      R_Coil( "DB8000_PART_STATUS".UNIT_02.FIXTURE_4.PART_A.STATUS.UNIT_02_STATUS.FACE_N_STATION_3_DONE )
   END_RUNG
   // the same network as SCL:
   IF "DB2430_FULL_DEPTH".FD_UNIT_02.FIXTURE_4.FD_STA_4_PULSE AND "DB8000_PART_STATUS".UNIT_02.FIXTURE_4.PART_A.STATUS.OK AND NOT "DB8000_PART_STATUS".UNIT_02.FIXTURE_4.PART_A.STATUS.PART_REJECTED THEN
       "DB8000_PART_STATUS".UNIT_02.FIXTURE_4.PART_A.STATUS.UNIT_02_STATUS.FACE_N_STATION_4_DONE := TRUE;
       "DB8000_PART_STATUS".UNIT_02.FIXTURE_4.PART_A.STATUS.UNIT_02_STATUS.FACE_N_STATION_3_DONE := FALSE;
   END_IF;
END_REGION

REGION Network 47: UNIT 02 FIXTURE 4 TOTAL FULL DEPTH / FULL DEPTH PULSE
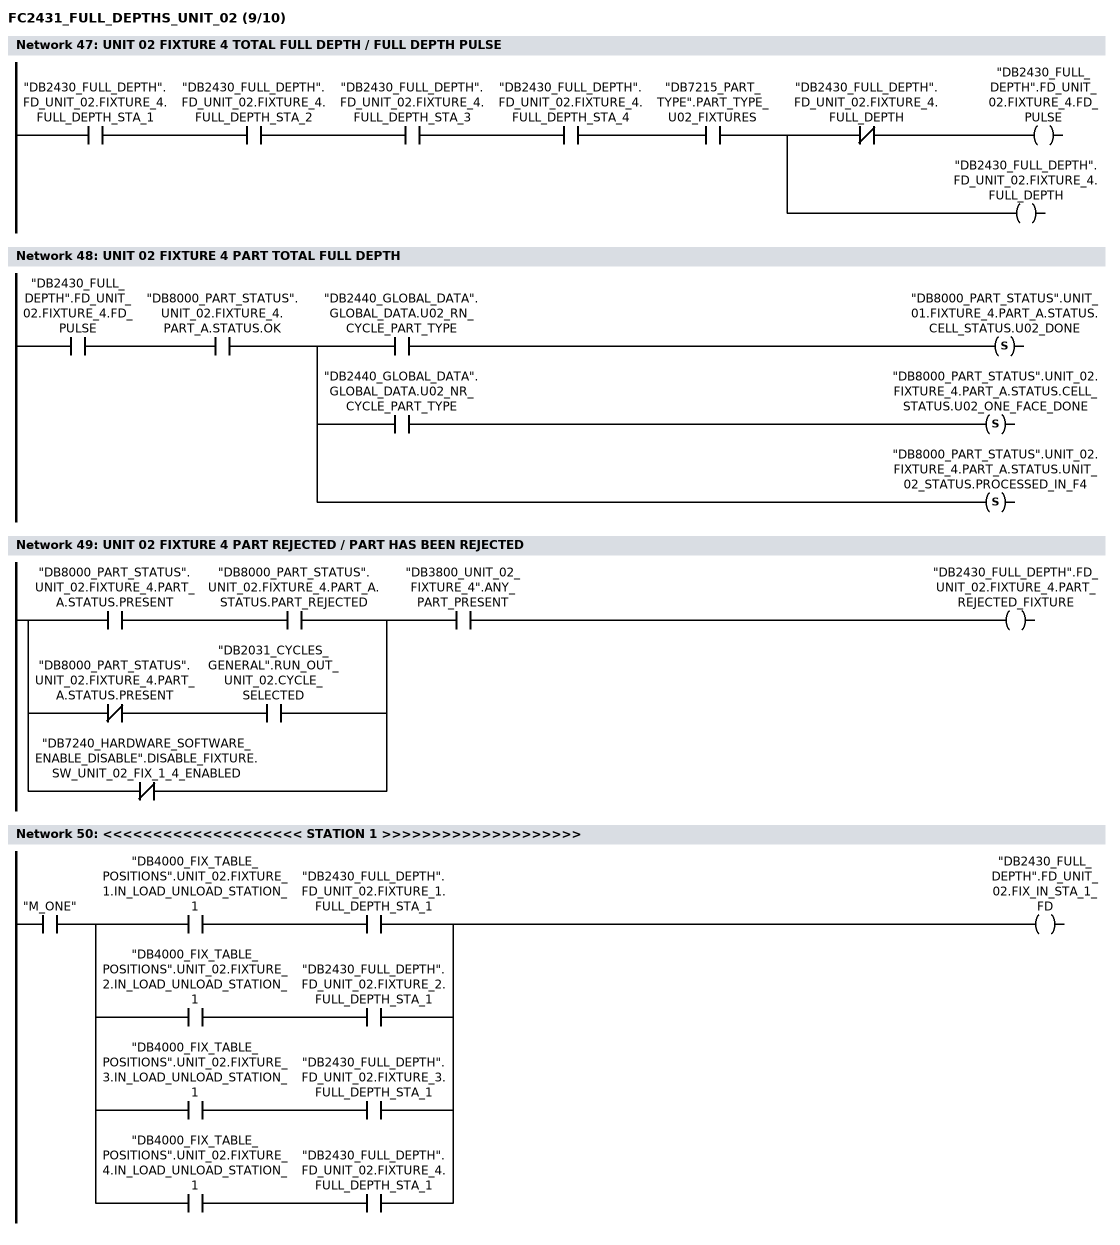
   RUNG wire#powerrail
      Contact( "DB2430_FULL_DEPTH".FD_UNIT_02.FIXTURE_4.FULL_DEPTH_STA_1 )
      Contact( "DB2430_FULL_DEPTH".FD_UNIT_02.FIXTURE_4.FULL_DEPTH_STA_2 )
      Contact( "DB2430_FULL_DEPTH".FD_UNIT_02.FIXTURE_4.FULL_DEPTH_STA_3 )
      Contact( "DB2430_FULL_DEPTH".FD_UNIT_02.FIXTURE_4.FULL_DEPTH_STA_4 )
      Contact( "DB7215_PART_TYPE".PART_TYPE_U02_FIXTURES )
      wire#w1
      I_Contact( "DB2430_FULL_DEPTH".FD_UNIT_02.FIXTURE_4.FULL_DEPTH )
      Coil( "DB2430_FULL_DEPTH".FD_UNIT_02.FIXTURE_4.FD_PULSE )
   END_RUNG
   RUNG wire#w1
      Coil( "DB2430_FULL_DEPTH".FD_UNIT_02.FIXTURE_4.FULL_DEPTH )
   END_RUNG
   // the same network as SCL:
   #_w1 := "DB2430_FULL_DEPTH".FD_UNIT_02.FIXTURE_4.FULL_DEPTH_STA_1 AND "DB2430_FULL_DEPTH".FD_UNIT_02.FIXTURE_4.FULL_DEPTH_STA_2 AND "DB2430_FULL_DEPTH".FD_UNIT_02.FIXTURE_4.FULL_DEPTH_STA_3 AND "DB2430_FULL_DEPTH".FD_UNIT_02.FIXTURE_4.FULL_DEPTH_STA_4 AND "DB7215_PART_TYPE".PART_TYPE_U02_FIXTURES;
   "DB2430_FULL_DEPTH".FD_UNIT_02.FIXTURE_4.FD_PULSE := #_w1 AND NOT "DB2430_FULL_DEPTH".FD_UNIT_02.FIXTURE_4.FULL_DEPTH;
   "DB2430_FULL_DEPTH".FD_UNIT_02.FIXTURE_4.FULL_DEPTH := #_w1;
END_REGION

REGION Network 48: UNIT 02 FIXTURE 4 PART TOTAL FULL DEPTH
   RUNG wire#powerrail
      Contact( "DB2430_FULL_DEPTH".FD_UNIT_02.FIXTURE_4.FD_PULSE )
      Contact( "DB8000_PART_STATUS".UNIT_02.FIXTURE_4.PART_A.STATUS.OK )
      wire#w1
      Contact( "DB2440_GLOBAL_DATA".GLOBAL_DATA.U02_RN_CYCLE_PART_TYPE )
      S_Coil( "DB8000_PART_STATUS".UNIT_01.FIXTURE_4.PART_A.STATUS.CELL_STATUS.U02_DONE )
   END_RUNG
   RUNG wire#w1
      Contact( "DB2440_GLOBAL_DATA".GLOBAL_DATA.U02_NR_CYCLE_PART_TYPE )
      S_Coil( "DB8000_PART_STATUS".UNIT_02.FIXTURE_4.PART_A.STATUS.CELL_STATUS.U02_ONE_FACE_DONE )
   END_RUNG
   RUNG wire#w1
      S_Coil( "DB8000_PART_STATUS".UNIT_02.FIXTURE_4.PART_A.STATUS.UNIT_02_STATUS.PROCESSED_IN_F4 )
   END_RUNG
   // the same network as SCL:
   #_w1 := "DB2430_FULL_DEPTH".FD_UNIT_02.FIXTURE_4.FD_PULSE AND "DB8000_PART_STATUS".UNIT_02.FIXTURE_4.PART_A.STATUS.OK;
   IF #_w1 AND "DB2440_GLOBAL_DATA".GLOBAL_DATA.U02_RN_CYCLE_PART_TYPE THEN
       "DB8000_PART_STATUS".UNIT_01.FIXTURE_4.PART_A.STATUS.CELL_STATUS.U02_DONE := TRUE;
   END_IF;
   IF #_w1 AND "DB2440_GLOBAL_DATA".GLOBAL_DATA.U02_NR_CYCLE_PART_TYPE THEN
       "DB8000_PART_STATUS".UNIT_02.FIXTURE_4.PART_A.STATUS.CELL_STATUS.U02_ONE_FACE_DONE := TRUE;
   END_IF;
   IF #_w1 THEN
       "DB8000_PART_STATUS".UNIT_02.FIXTURE_4.PART_A.STATUS.UNIT_02_STATUS.PROCESSED_IN_F4 := TRUE;
   END_IF;
END_REGION

REGION Network 49: UNIT 02 FIXTURE 4 PART REJECTED / PART HAS BEEN REJECTED
   RUNG wire#powerrail
      Contact( "DB8000_PART_STATUS".UNIT_02.FIXTURE_4.PART_A.STATUS.PRESENT )
      Contact( "DB8000_PART_STATUS".UNIT_02.FIXTURE_4.PART_A.STATUS.PART_REJECTED )
      wire#w1
      Contact( "DB3800_UNIT_02_FIXTURE_4".ANY_PART_PRESENT )
      Coil( "DB2430_FULL_DEPTH".FD_UNIT_02.FIXTURE_4.PART_REJECTED_FIXTURE )
   END_RUNG
   RUNG wire#powerrail
      I_Contact( "DB8000_PART_STATUS".UNIT_02.FIXTURE_4.PART_A.STATUS.PRESENT )
      Contact( "DB2031_CYCLES_GENERAL".RUN_OUT_UNIT_02.CYCLE_SELECTED )
   END_RUNG wire#w1
   RUNG wire#powerrail
      I_Contact( "DB7240_HARDWARE_SOFTWARE_ENABLE_DISABLE".DISABLE_FIXTURE.SW_UNIT_02_FIX_1_4_ENABLED )
   END_RUNG wire#w1
   // the same network as SCL:
   "DB2430_FULL_DEPTH".FD_UNIT_02.FIXTURE_4.PART_REJECTED_FIXTURE := (("DB8000_PART_STATUS".UNIT_02.FIXTURE_4.PART_A.STATUS.PRESENT AND "DB8000_PART_STATUS".UNIT_02.FIXTURE_4.PART_A.STATUS.PART_REJECTED) OR (NOT "DB8000_PART_STATUS".UNIT_02.FIXTURE_4.PART_A.STATUS.PRESENT AND "DB2031_CYCLES_GENERAL".RUN_OUT_UNIT_02.CYCLE_SELECTED) OR NOT "DB7240_HARDWARE_SOFTWARE_ENABLE_DISABLE".DISABLE_FIXTURE.SW_UNIT_02_FIX_1_4_ENABLED) AND "DB3800_UNIT_02_FIXTURE_4".ANY_PART_PRESENT;
END_REGION

REGION Network 50: <<<<<<<<<<<<<<<<<<<< STATION 1 >>>>>>>>>>>>>>>>>>>>
   RUNG wire#powerrail
      Contact( "M_ONE" )
      wire#w1
      Contact( "DB4000_FIX_TABLE_POSITIONS".UNIT_02.FIXTURE_1.IN_LOAD_UNLOAD_STATION_1 )
      Contact( "DB2430_FULL_DEPTH".FD_UNIT_02.FIXTURE_1.FULL_DEPTH_STA_1 )
      wire#w2
      Coil( "DB2430_FULL_DEPTH".FD_UNIT_02.FIX_IN_STA_1_FD )
   END_RUNG
   RUNG wire#w1
      Contact( "DB4000_FIX_TABLE_POSITIONS".UNIT_02.FIXTURE_2.IN_LOAD_UNLOAD_STATION_1 )
      Contact( "DB2430_FULL_DEPTH".FD_UNIT_02.FIXTURE_2.FULL_DEPTH_STA_1 )
   END_RUNG wire#w2
   RUNG wire#w1
      Contact( "DB4000_FIX_TABLE_POSITIONS".UNIT_02.FIXTURE_3.IN_LOAD_UNLOAD_STATION_1 )
      Contact( "DB2430_FULL_DEPTH".FD_UNIT_02.FIXTURE_3.FULL_DEPTH_STA_1 )
   END_RUNG wire#w2
   RUNG wire#w1
      Contact( "DB4000_FIX_TABLE_POSITIONS".UNIT_02.FIXTURE_4.IN_LOAD_UNLOAD_STATION_1 )
      Contact( "DB2430_FULL_DEPTH".FD_UNIT_02.FIXTURE_4.FULL_DEPTH_STA_1 )
   END_RUNG wire#w2
   // the same network as SCL:
   "DB2430_FULL_DEPTH".FD_UNIT_02.FIX_IN_STA_1_FD := "M_ONE" AND (("DB4000_FIX_TABLE_POSITIONS".UNIT_02.FIXTURE_1.IN_LOAD_UNLOAD_STATION_1 AND "DB2430_FULL_DEPTH".FD_UNIT_02.FIXTURE_1.FULL_DEPTH_STA_1) OR ("DB4000_FIX_TABLE_POSITIONS".UNIT_02.FIXTURE_2.IN_LOAD_UNLOAD_STATION_1 AND "DB2430_FULL_DEPTH".FD_UNIT_02.FIXTURE_2.FULL_DEPTH_STA_1) OR ("DB4000_FIX_TABLE_POSITIONS".UNIT_02.FIXTURE_3.IN_LOAD_UNLOAD_STATION_1 AND "DB2430_FULL_DEPTH".FD_UNIT_02.FIXTURE_3.FULL_DEPTH_STA_1) OR ("DB4000_FIX_TABLE_POSITIONS".UNIT_02.FIXTURE_4.IN_LOAD_UNLOAD_STATION_1 AND "DB2430_FULL_DEPTH".FD_UNIT_02.FIXTURE_4.FULL_DEPTH_STA_1));
END_REGION

REGION Network 51: <<<<<<<<<<<<<<<<<<<< STATION 2 >>>>>>>>>>>>>>>>>>>>
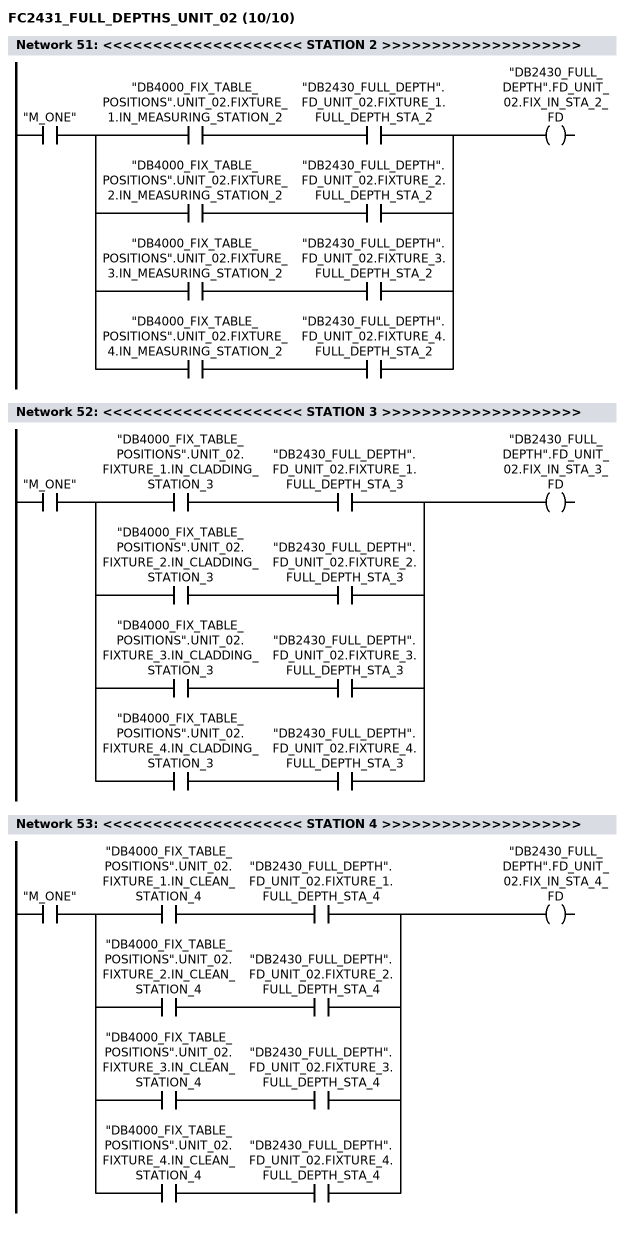
   RUNG wire#powerrail
      Contact( "M_ONE" )
      wire#w1
      Contact( "DB4000_FIX_TABLE_POSITIONS".UNIT_02.FIXTURE_1.IN_MEASURING_STATION_2 )
      Contact( "DB2430_FULL_DEPTH".FD_UNIT_02.FIXTURE_1.FULL_DEPTH_STA_2 )
      wire#w2
      Coil( "DB2430_FULL_DEPTH".FD_UNIT_02.FIX_IN_STA_2_FD )
   END_RUNG
   RUNG wire#w1
      Contact( "DB4000_FIX_TABLE_POSITIONS".UNIT_02.FIXTURE_2.IN_MEASURING_STATION_2 )
      Contact( "DB2430_FULL_DEPTH".FD_UNIT_02.FIXTURE_2.FULL_DEPTH_STA_2 )
   END_RUNG wire#w2
   RUNG wire#w1
      Contact( "DB4000_FIX_TABLE_POSITIONS".UNIT_02.FIXTURE_3.IN_MEASURING_STATION_2 )
      Contact( "DB2430_FULL_DEPTH".FD_UNIT_02.FIXTURE_3.FULL_DEPTH_STA_2 )
   END_RUNG wire#w2
   RUNG wire#w1
      Contact( "DB4000_FIX_TABLE_POSITIONS".UNIT_02.FIXTURE_4.IN_MEASURING_STATION_2 )
      Contact( "DB2430_FULL_DEPTH".FD_UNIT_02.FIXTURE_4.FULL_DEPTH_STA_2 )
   END_RUNG wire#w2
   // the same network as SCL:
   "DB2430_FULL_DEPTH".FD_UNIT_02.FIX_IN_STA_2_FD := "M_ONE" AND (("DB4000_FIX_TABLE_POSITIONS".UNIT_02.FIXTURE_1.IN_MEASURING_STATION_2 AND "DB2430_FULL_DEPTH".FD_UNIT_02.FIXTURE_1.FULL_DEPTH_STA_2) OR ("DB4000_FIX_TABLE_POSITIONS".UNIT_02.FIXTURE_2.IN_MEASURING_STATION_2 AND "DB2430_FULL_DEPTH".FD_UNIT_02.FIXTURE_2.FULL_DEPTH_STA_2) OR ("DB4000_FIX_TABLE_POSITIONS".UNIT_02.FIXTURE_3.IN_MEASURING_STATION_2 AND "DB2430_FULL_DEPTH".FD_UNIT_02.FIXTURE_3.FULL_DEPTH_STA_2) OR ("DB4000_FIX_TABLE_POSITIONS".UNIT_02.FIXTURE_4.IN_MEASURING_STATION_2 AND "DB2430_FULL_DEPTH".FD_UNIT_02.FIXTURE_4.FULL_DEPTH_STA_2));
END_REGION

REGION Network 52: <<<<<<<<<<<<<<<<<<<< STATION 3 >>>>>>>>>>>>>>>>>>>>
   RUNG wire#powerrail
      Contact( "M_ONE" )
      wire#w1
      Contact( "DB4000_FIX_TABLE_POSITIONS".UNIT_02.FIXTURE_1.IN_CLADDING_STATION_3 )
      Contact( "DB2430_FULL_DEPTH".FD_UNIT_02.FIXTURE_1.FULL_DEPTH_STA_3 )
      wire#w2
      Coil( "DB2430_FULL_DEPTH".FD_UNIT_02.FIX_IN_STA_3_FD )
   END_RUNG
   RUNG wire#w1
      Contact( "DB4000_FIX_TABLE_POSITIONS".UNIT_02.FIXTURE_2.IN_CLADDING_STATION_3 )
      Contact( "DB2430_FULL_DEPTH".FD_UNIT_02.FIXTURE_2.FULL_DEPTH_STA_3 )
   END_RUNG wire#w2
   RUNG wire#w1
      Contact( "DB4000_FIX_TABLE_POSITIONS".UNIT_02.FIXTURE_3.IN_CLADDING_STATION_3 )
      Contact( "DB2430_FULL_DEPTH".FD_UNIT_02.FIXTURE_3.FULL_DEPTH_STA_3 )
   END_RUNG wire#w2
   RUNG wire#w1
      Contact( "DB4000_FIX_TABLE_POSITIONS".UNIT_02.FIXTURE_4.IN_CLADDING_STATION_3 )
      Contact( "DB2430_FULL_DEPTH".FD_UNIT_02.FIXTURE_4.FULL_DEPTH_STA_3 )
   END_RUNG wire#w2
   // the same network as SCL:
   "DB2430_FULL_DEPTH".FD_UNIT_02.FIX_IN_STA_3_FD := "M_ONE" AND (("DB4000_FIX_TABLE_POSITIONS".UNIT_02.FIXTURE_1.IN_CLADDING_STATION_3 AND "DB2430_FULL_DEPTH".FD_UNIT_02.FIXTURE_1.FULL_DEPTH_STA_3) OR ("DB4000_FIX_TABLE_POSITIONS".UNIT_02.FIXTURE_2.IN_CLADDING_STATION_3 AND "DB2430_FULL_DEPTH".FD_UNIT_02.FIXTURE_2.FULL_DEPTH_STA_3) OR ("DB4000_FIX_TABLE_POSITIONS".UNIT_02.FIXTURE_3.IN_CLADDING_STATION_3 AND "DB2430_FULL_DEPTH".FD_UNIT_02.FIXTURE_3.FULL_DEPTH_STA_3) OR ("DB4000_FIX_TABLE_POSITIONS".UNIT_02.FIXTURE_4.IN_CLADDING_STATION_3 AND "DB2430_FULL_DEPTH".FD_UNIT_02.FIXTURE_4.FULL_DEPTH_STA_3));
END_REGION

REGION Network 53: <<<<<<<<<<<<<<<<<<<< STATION 4 >>>>>>>>>>>>>>>>>>>>
   RUNG wire#powerrail
      Contact( "M_ONE" )
      wire#w1
      Contact( "DB4000_FIX_TABLE_POSITIONS".UNIT_02.FIXTURE_1.IN_CLEAN_STATION_4 )
      Contact( "DB2430_FULL_DEPTH".FD_UNIT_02.FIXTURE_1.FULL_DEPTH_STA_4 )
      wire#w2
      Coil( "DB2430_FULL_DEPTH".FD_UNIT_02.FIX_IN_STA_4_FD )
   END_RUNG
   RUNG wire#w1
      Contact( "DB4000_FIX_TABLE_POSITIONS".UNIT_02.FIXTURE_2.IN_CLEAN_STATION_4 )
      Contact( "DB2430_FULL_DEPTH".FD_UNIT_02.FIXTURE_2.FULL_DEPTH_STA_4 )
   END_RUNG wire#w2
   RUNG wire#w1
      Contact( "DB4000_FIX_TABLE_POSITIONS".UNIT_02.FIXTURE_3.IN_CLEAN_STATION_4 )
      Contact( "DB2430_FULL_DEPTH".FD_UNIT_02.FIXTURE_3.FULL_DEPTH_STA_4 )
   END_RUNG wire#w2
   RUNG wire#w1
      Contact( "DB4000_FIX_TABLE_POSITIONS".UNIT_02.FIXTURE_4.IN_CLEAN_STATION_4 )
      Contact( "DB2430_FULL_DEPTH".FD_UNIT_02.FIXTURE_4.FULL_DEPTH_STA_4 )
   END_RUNG wire#w2
   // the same network as SCL:
   "DB2430_FULL_DEPTH".FD_UNIT_02.FIX_IN_STA_4_FD := "M_ONE" AND (("DB4000_FIX_TABLE_POSITIONS".UNIT_02.FIXTURE_1.IN_CLEAN_STATION_4 AND "DB2430_FULL_DEPTH".FD_UNIT_02.FIXTURE_1.FULL_DEPTH_STA_4) OR ("DB4000_FIX_TABLE_POSITIONS".UNIT_02.FIXTURE_2.IN_CLEAN_STATION_4 AND "DB2430_FULL_DEPTH".FD_UNIT_02.FIXTURE_2.FULL_DEPTH_STA_4) OR ("DB4000_FIX_TABLE_POSITIONS".UNIT_02.FIXTURE_3.IN_CLEAN_STATION_4 AND "DB2430_FULL_DEPTH".FD_UNIT_02.FIXTURE_3.FULL_DEPTH_STA_4) OR ("DB4000_FIX_TABLE_POSITIONS".UNIT_02.FIXTURE_4.IN_CLEAN_STATION_4 AND "DB2430_FULL_DEPTH".FD_UNIT_02.FIXTURE_4.FULL_DEPTH_STA_4));
END_REGION
END_FUNCTION
